(* CODESYS project BasePpt.library
   Company: Vistaprint
   Title: BasePpt
   Description: 0.0.0.10 - PCE: no EOFF State!! in EOFF go to OFF (in Always); Redo changes of 0.0.0.6; PTS.Always no EOFF; sta_OFFBusy in PTS reworked;
      0.0.0.9 - Merged the DeStacker MDC with the BasePpt MDC
      0.0.0.8 - Added newer Versions of libraries.
      0.0.0.7 - Added newer Versions of libraries.
      0.0.0.6 - Changes for Simualtion in MDC, sta_OFFBusy in PTB/MDC reworked; Always in PTB reworked;
      0.0.0.5 - Added new Base_PLC 0.3.4.1
      0.0.0.4 - Bug fixed in FB_PTB
      0.0.0.3 - Update to take the newest libraries 
      0.0.0.2 - Update to Base_PLC 0.3.3.2; Update to Base_Elements 0.0.0.9
   Author: pcipriano
   Version: 0.0.0.10

Project tree, tasks and I/O mapping:
  libraries: Base_Elements, 0.0.1.4 (Vistaprint); Base_PLC, 0.3.4.3 (Vistaprint); Tc2_Standard, 3.3.0.0 (Beckhoff Automation GmbH); Tc2_System, * (Beckhoff Automation GmbH); Tc2_Utilities, * (Beckhoff Automation GmbH); Tc3_Interfaces, 3.3.0.0 (Beckhoff Automation GmbH); Tc3_Module, * (Beckhoff Automation GmbH)
  POUs/
    Controller/
      Driver/
        PTR [Paper Tracker]/
          data type E_PTR_Status
          function block FB_PTR [ST]: BeltLength, EnterComplete, FB_init, Insert, PaperEntryOffset, PaperOnBelt, Pop, PositionList, Push, Reset, TimeBase
          data type T_PTR_STRUCT
      Lvl0/
      Lvl1/
        MDC [Malteser Drive Controller]/
          data type E_ALM_MDC
          function block FB_MDC [ST]: ActualPosition, Always, CtrlInit, CtrlSIf, Drive, FB_init, getCmdState, getCtrlSIf, GetTurningDirection, IncrementPosition, IoInBridge, IoOutBridge, SetPositionToGo, sta_ERROR, sta_ERRORQuit, sta_InitializeBusy, sta_InPosition, sta_InPositionBusy, sta_OFF, sta_OFFBusy, sta_PON, sta_PREPOSITION, sta_PREPOSITIONbusy, sta_StartTurnBusy, sta_TurnBusy, sta_TURNDONE, StateMachine
          global variables MDC_CmdState
          data type T_Ctrl_SIf_MDC
          data type T_Ctrl_SIf_MDC_Cfg
          data type T_Ctrl_SIf_MDC_Cur
          data type T_Ctrl_SIf_MDC_Ilk
          data type T_Ctrl_SIf_MDC_In
          data type T_Ctrl_SIf_MDC_Out
          data type T_Ctrl_SIf_MDC_Par
        PTB [Paper Transport Belt]/
          BeltParameterFunction/
            data type T_Belt_Cfg_Base
            data type T_Belt_Cur_Base
            data type T_Belt_Par_Base
          data type E_ALM_PTB
          data type E_BELT_DIRECTION
          data type E_PTB_MODE
          data type E_PTB_PaperDirection
          function block FB_PTB [ST]: Always, CalculateBeltParameter, CalculateModeParameter, CheckPumpState, cmd_OFF, cmd_RUN, cmd_STOP, CtrlInit, CtrlSIf, Drive, FB_init, getCmdState, getCtrlSIf, IoInBridge, IoOutBridge, PaperPositionHandling, PositionList, SetPumpComand, sta_EJECTPAPER, sta_EJECTPAPERbusy, sta_ERROR, sta_ERRORQuit, sta_OFF, sta_OFFBusy, sta_PON, sta_RUN, sta_RUNBusy, sta_STACKPAPER, sta_STACKPAPERbusy, sta_STOP, sta_STOPBusy, StateMachine, VacuumPump
          global variables PTB_CmdState
          data type T_Ctrl_SIf_PTB
          data type T_Ctrl_SIf_PTB_Cfg
          data type T_Ctrl_SIf_PTB_Cur
          data type T_Ctrl_SIf_PTB_Ilk
          data type T_Ctrl_SIf_PTB_In
          data type T_Ctrl_SIf_PTB_Out
          data type T_Ctrl_SIf_PTB_Par
      Lvl2/
        PBC [Paper Buffer Controller]/
          data type E_ALM_PBC
          function block FB_PBC [ST]: Always, Belt, CountPaper, CtrlInit, CtrlSIf, DeStacker, FB_init, getCmdState, getCtrlSIf, IoInBridge, IoOutBridge, PaperHight, PaperWidth, sta_EjectBusy, sta_EjectCheck, sta_ERROR, sta_ERRORQuit, sta_OFF, sta_OFFBusy, sta_PON, sta_PositionPaperBusy, sta_RUN, sta_RUNbusy, sta_STANDBY, sta_STANDBYBusy, StateMachine
          global variables PBC_CmdState
          data type T_Ctrl_SIf_PBC
          data type T_Ctrl_SIf_PBC_Cfg
          data type T_Ctrl_SIf_PBC_Cur
          data type T_Ctrl_SIf_PBC_Ilk
          data type T_Ctrl_SIf_PBC_In
          data type T_Ctrl_SIf_PBC_Out
          data type T_Ctrl_SIf_PBC_Par
        PCE [Paper Belt Corner Element]/
          data type E_ALM_PCE
          function block FB_PCE [ST]: Always, CtrlInit, CtrlSIf, DriveIn, DriveOut, FB_init, getCmdState, IoInBridge, IoOutBridge, PaperExitValveActive, PaperInputValveActive, sta_ERROR, sta_ERRORQuit, sta_OFF, sta_OFFBusy, sta_PON, sta_RUN, sta_RUNBusy, sta_STOP, sta_STOPBusy, StateMachine
          global variables PCE_CmdState
          data type T_Ctrl_SIf_PCE
          data type T_Ctrl_SIf_PCE_Cfg
          data type T_Ctrl_SIf_PCE_Cur
          data type T_Ctrl_SIf_PCE_Ilk
          data type T_Ctrl_SIf_PCE_In
          data type T_Ctrl_SIf_PCE_Out
          data type T_Ctrl_SIf_PCE_Par
      Lvl3/
        PTS [Paper Turning Station]/
          data type E_ALM_PTS
          data type E_PTS_MODE
          function block FB_PTS [ST]: Always, Belt, CalculateOutputDelay, CtrlInit, CtrlSIf, FB_init, getCmdState, getCtrlSIf, GetItemBusy, IoInBridge, IoOutBridge, Malteser, sta_EmptyDelayBusy, sta_ERROR, sta_ERRORQuit, sta_GetItemBusy, sta_InitializeBusy, sta_OFF, sta_OFFBusy, sta_PaperDelayBusy, sta_PON, sta_RUN, sta_RUNBusy, sta_STANDBY, sta_STANDBYBusy, sta_STOP, sta_STOPbusy, sta_TurnEmptyBusy, sta_TurnPaperBusy, sta_WaitPaper, sta_WaitPaperGone, StateMachine
          global variables PTS_CmdState
          data type T_Ctrl_SIf_PTS
          data type T_Ctrl_SIf_PTS_Cfg
          data type T_Ctrl_SIf_PTS_Cur
          data type T_Ctrl_SIf_PTS_Ilk
          data type T_Ctrl_SIf_PTS_In
          data type T_Ctrl_SIf_PTS_Out
          data type T_Ctrl_SIf_PTS_Par
          data type T_PTS_InOutPositions
      Lvl4/
      Top/
  Version/
    global variables Global_Version
*)

// POUs/Controller/Driver/PTR [Paper Tracker]/E_PTR_Status
TYPE E_PTR_Status :
(
	EnterBusy,
	OnBelt,
	ExitBusy,
	Gone,
	ERROR,
	MAX_E_PTR_Status
);
END_TYPE

// POUs/Controller/Driver/PTR [Paper Tracker]/T_PTR_STRUCT
TYPE T_PTR_STRUCT :
STRUCT
	// [us] Time of the paper on the belt
	udiTimeOnBelt_us				: UDINT;
	// [mm] Position of the paper on the belt
	lrePositionOnBelt_mm			: LREAL;
	// [mm] Position of the paper on the belt Adjusted to the possible maximum
	lrePositionOnBeltAdjusted_mm	: LREAL;
	// Paper Item Id
	udiItemId						: UDINT;
	// Error	
	eStatus							: E_PTR_Status;
END_STRUCT
END_TYPE

// POUs/Controller/Lvl1/MDC [Malteser Drive Controller]/E_ALM_MDC
TYPE E_ALM_MDC :
(
	TableSensorTimeout 		:= 1,
	CrossSensorTimeout		:= 2,
	PositionSame			:= 3,
	MAX_E_ALM_MDC
);
END_TYPE

// POUs/Controller/Lvl1/MDC [Malteser Drive Controller]/T_Ctrl_SIf_MDC
TYPE T_Ctrl_SIf_MDC :
STRUCT
	///configuration
	Cfg: T_Ctrl_SIf_MDC_Cfg;
	///parameter
	Par: T_Ctrl_SIf_MDC_Par;
	///current values
	Cur: T_Ctrl_SIf_MDC_Cur;
	///io input
	In: T_Ctrl_SIf_MDC_In;
	///io output
	Out: T_Ctrl_SIf_MDC_Out;
	///alarm number used in this controller
	Alm: ARRAY[1..MAX_E_ALM_MDC] OF T_Ctrl_Alm;
	///interlock of output/movements
	Ilk: T_Ctrl_SIf_MDC_Ilk;
END_STRUCT
END_TYPE

// POUs/Controller/Lvl1/MDC [Malteser Drive Controller]/T_Ctrl_SIf_MDC_Cfg
TYPE T_Ctrl_SIf_MDC_Cfg :
STRUCT
	/// Number of positions in 360° of the Malteser drive
	uintPositionPerTurn		: UINT;
END_STRUCT
END_TYPE

// POUs/Controller/Lvl1/MDC [Malteser Drive Controller]/T_Ctrl_SIf_MDC_Cur
TYPE T_Ctrl_SIf_MDC_Cur :
STRUCT	
	/// Actual Position as position 
	uintActualPosition			: UINT;
	/// actual turning direction
	eActualTurningDirection		: E_TURN_DIRECTION;
	/// Reference still ok
	bolReferenceOk				: BOOL;		
END_STRUCT
END_TYPE

// POUs/Controller/Lvl1/MDC [Malteser Drive Controller]/T_Ctrl_SIf_MDC_Ilk
TYPE T_Ctrl_SIf_MDC_Ilk :
STRUCT
END_STRUCT
END_TYPE

// POUs/Controller/Lvl1/MDC [Malteser Drive Controller]/T_Ctrl_SIf_MDC_In
TYPE T_Ctrl_SIf_MDC_In :
STRUCT
	/// Is the cross in sensor positinon. One rotation step done.
	bolCrossPositionSensor				: BASE_PLC.T_Ctrl_IoBool;
	/// Is the table at 0° degrees
	bolTablePositionSensor				: BASE_PLC.T_Ctrl_IoBool;
END_STRUCT
END_TYPE

// POUs/Controller/Lvl1/MDC [Malteser Drive Controller]/T_Ctrl_SIf_MDC_Out
TYPE T_Ctrl_SIf_MDC_Out :
STRUCT
	intActualPosition		: BASE_PLC.T_Ctrl_IoInt;
END_STRUCT
END_TYPE

// POUs/Controller/Lvl1/MDC [Malteser Drive Controller]/T_Ctrl_SIf_MDC_Par
TYPE T_Ctrl_SIf_MDC_Par :
STRUCT
	/// <0 = Turn left; =0 automatic; >0 turn right
	intTurnDirection					: INT;
	/// Position to go to if comand turn is given. 0 = initialization position
	uinPositionToGo						: UINT;
	/// [ms] time to rotate one step 
	udiStepRotationTime_ms				: UDINT;
	/// [ms] initialization timeout time
	udiInitializationTime_ms			: UDINT;
	/// [ms] simulation time to rotate one step
	udiSimStepRotationTime_ms			: UDINT;
	/// [ms] simulation initialization timeout time
	udiSimInitializationTime_ms			: UDINT;
	/// [ms] simulation time to start rotate and Cross sensor needs to go away
	udiSimStartRotationTime_ms			: UDINT;
	/// [rpm] PrePosition Speed
	uinPrePositionSpeed_rpm				: UINT;
	/// [rpm] Position Speed
	uinPositionSpeed_rpm				: UINT;
END_STRUCT
END_TYPE

// POUs/Controller/Lvl1/PTB [Paper Transport Belt]/BeltParameterFunction/T_Belt_Cfg_Base
TYPE T_Belt_Cfg_Base :
STRUCT
	/// Assign the motor rotation to a belt direction.
	intForwardDirection				: INT;
	/// Assign the motor rotation to a belt direction.
	intBackwardDirection			: INT;
	/// [mm] the belt travels per motor rotation
	reaRpmDistance_mm					: REAL;
END_STRUCT
END_TYPE

// POUs/Controller/Lvl1/PTB [Paper Transport Belt]/BeltParameterFunction/T_Belt_Cur_Base
TYPE T_Belt_Cur_Base :
STRUCT
	/// [mm/s] Belt speed
	uinBeltSpeed_mms						: UINT;
	/// [rpm] Belt speed
	uinBeltSpeed_rpm						: UINT;
END_STRUCT
END_TYPE

// POUs/Controller/Lvl1/PTB [Paper Transport Belt]/BeltParameterFunction/T_Belt_Par_Base
TYPE T_Belt_Par_Base :
STRUCT
	/// eSpeedControlSelection.EFFECTIVE_SPEED : [mm/sec] Target speed. Uses reaRpmDistance_mm and uinLC11 to calculate the rpm
	uinBeltSpeed						: UINT;
	/// eSpeedControlSelection.EFFECTIVE_SPEED : [mm/sec] Target speed. Uses reaRpmDistance_mm and uinLC11 to calculate the rpm
	uinStackSpeed						: UINT;
END_STRUCT
END_TYPE

// POUs/Controller/Lvl1/PTB [Paper Transport Belt]/E_ALM_PTB
TYPE E_ALM_PTB :
(
	TestAlarm := 1,
	MAX_E_ALM_PTB 
);
END_TYPE

// POUs/Controller/Lvl1/PTB [Paper Transport Belt]/E_BELT_DIRECTION
TYPE E_BELT_DIRECTION :
(
	FORWARD			:= 0,
	BACKWARD		:= 1,
	MAX_E_BELT_DIRECTION
);
END_TYPE

// POUs/Controller/Lvl1/PTB [Paper Transport Belt]/E_PTB_MODE
TYPE E_PTB_MODE :
(
	Endless	,		// 0
	ToSensor,		// 1
	ToDistance,		// 2
	ToTime,			// 3
	Stack,			// 4
	MAX_E_PTB_MODE
);
END_TYPE

// POUs/Controller/Lvl1/PTB [Paper Transport Belt]/E_PTB_PaperDirection
TYPE E_PTB_PaperDirection :
(
	Portrait,
	Landscape,
	MAX_E_PTB_PaperDirection
);
END_TYPE

// POUs/Controller/Lvl1/PTB [Paper Transport Belt]/T_Ctrl_SIf_PTB
TYPE T_Ctrl_SIf_PTB :
STRUCT
	///configuration
	Cfg: T_Ctrl_SIf_PTB_Cfg;
	///parameter
	Par: T_Ctrl_SIf_PTB_Par;
	///current values
	Cur: T_Ctrl_SIf_PTB_Cur;
	///io input
	In: T_Ctrl_SIf_PTB_In;
	///io output
	Out: T_Ctrl_SIf_PTB_Out;
	///alarm number used in this controller
	Alm: ARRAY[1..E_ALM_PTB.MAX_E_ALM_PTB] OF T_Ctrl_Alm;
	///interlock of output/movements
	Ilk: T_Ctrl_SIf_PTB_Ilk;
END_STRUCT
END_TYPE

// POUs/Controller/Lvl1/PTB [Paper Transport Belt]/T_Ctrl_SIf_PTB_Cfg
TYPE T_Ctrl_SIf_PTB_Cfg :
STRUCT
	// Function Mode
	eMode							: E_PTB_MODE;
	// Vacuum pump present
	bolVacuumPresent				: BOOL;
	// [mm] Length of the belt
	udiBeltLength_mm				: UDINT;
	// Belt Parameter	
	rBeltParam						: T_Belt_Cfg_Base;
	// Enable Entry Belt Sensor Debounce
	bolEntrySensorDebounceEnable	: BOOL;
	// Enable Exit Belt Sensor Debounce
	bolExitSensorDebounceEnable		: BOOL;
END_STRUCT
END_TYPE

// POUs/Controller/Lvl1/PTB [Paper Transport Belt]/T_Ctrl_SIf_PTB_Cur
	TYPE T_Ctrl_SIf_PTB_Cur :
STRUCT	
	/// actual belt direction
	eActualDirection						: E_BELT_DIRECTION;
	/// [mm] Distance to move if Move Mode is distance
	udiDistanceToMove_mm					: UDINT;
	/// [ms] Time to move
	udiTimeToMove_ms						: UDINT;
	// Belt parameter
	rBeltParam								: T_Belt_Cur_Base;
	// Belt Run Time
	udiBeltTimeBase_mm						: UDINT;
	// Paper on the belt
	uinPaperOnBelt							: UINT;
	// Pointer to the Position list of the paper on the belt
	pPositionList							: POINTER TO T_PTR_STRUCT;
END_STRUCT
END_TYPE

// POUs/Controller/Lvl1/PTB [Paper Transport Belt]/T_Ctrl_SIf_PTB_Ilk
TYPE T_Ctrl_SIf_PTB_Ilk :
STRUCT
END_STRUCT
END_TYPE

// POUs/Controller/Lvl1/PTB [Paper Transport Belt]/T_Ctrl_SIf_PTB_In
TYPE T_Ctrl_SIf_PTB_In :
STRUCT
	bolBeltEntrySensor			: BASE_PLC.T_Ctrl_IoBool;
	bolBeltExitSensor			: BASE_PLC.T_Ctrl_IoBool;
	bolBeltEntrySensorPEdge		: BASE_PLC.T_Ctrl_IoBool;
	bolBeltEntrySensorNEdge		: BASE_PLC.T_Ctrl_IoBool;
	bolBeltExitSensorPEdge		: BASE_PLC.T_Ctrl_IoBool;
	bolBeltExitSensorNEdge		: BASE_PLC.T_Ctrl_IoBool;
END_STRUCT
END_TYPE

// POUs/Controller/Lvl1/PTB [Paper Transport Belt]/T_Ctrl_SIf_PTB_Out
TYPE T_Ctrl_SIf_PTB_Out :
STRUCT

END_STRUCT
END_TYPE

// POUs/Controller/Lvl1/PTB [Paper Transport Belt]/T_Ctrl_SIf_PTB_Par
TYPE T_Ctrl_SIf_PTB_Par :
STRUCT
	/// <0 = Backward; =0 None; >0 forward
	intDirection						: INT;
	/// [mm] Distance to move if Move Mode is distance
	udiDistanceToMove_mm				: UDINT;
	/// [ms] Time to move
	udiTimeToMove_ms					: UDINT;
	/// Stack hight in # of sheets
	uinPaperStackHight					: UINT;
	/// Automatic ejecting the paper if stackhight is reached
	bolAutoEjectAfterStack				: BOOL;
	/// Automatic stacking the paper after ejecting all paper
	bolAutoStackAfterEject				: BOOL;
	/// Belt Parameter
	rBeltParam							: T_Belt_Par_Base;
	// [ms] Stack delay time - Delay before out motor can move after paper entered system
	udiStackDelayTime_ms				: UDINT;
	// [mm] Belt Length
	udiBeltLength_mm					: UDINT;
	// Page running format
	ePaperOrientation					: E_PTB_PaperDirection;
	/// [mm] Paper Hight
	uinPaperHight_mm					: UINT;
	/// [mm] Paper Width
	uinPaperWidth_mm					: UINT;
	// [ms] Input Parameter Debounce time
	uinInputSignalDebounceTime_ms		: UINT;
END_STRUCT
END_TYPE

// POUs/Controller/Lvl2/PBC [Paper Buffer Controller]/E_ALM_PBC
TYPE E_ALM_PBC :
(
	PaperTransport			:= 1,
	BufferFull				:= 2,
	BufferEmpty				:= 3,
	MAX_E_ALM_PBC
);
END_TYPE

// POUs/Controller/Lvl2/PBC [Paper Buffer Controller]/T_Ctrl_SIf_PBC
TYPE T_Ctrl_SIf_PBC :
STRUCT
	///configuration
	Cfg: T_Ctrl_SIf_PBC_Cfg;
	///parameter
	Par: T_Ctrl_SIf_PBC_Par;
	///current values
	Cur: T_Ctrl_SIf_PBC_Cur;
	///io input
	In: T_Ctrl_SIf_PBC_In;
	///io output
	Out: T_Ctrl_SIf_PBC_Out;
	///alarm number used in this controller
	Alm: ARRAY[1..E_ALM_PBC.MAX_E_ALM_PBC] OF T_Ctrl_Alm;
	///interlock of output/movements
	Ilk: T_Ctrl_SIf_PBC_Ilk;
END_STRUCT
END_TYPE

// POUs/Controller/Lvl2/PBC [Paper Buffer Controller]/T_Ctrl_SIf_PBC_Cfg
TYPE T_Ctrl_SIf_PBC_Cfg :
STRUCT
END_STRUCT
END_TYPE

// POUs/Controller/Lvl2/PBC [Paper Buffer Controller]/T_Ctrl_SIf_PBC_Cur
TYPE T_Ctrl_SIf_PBC_Cur :
STRUCT	
	/// How many papers are in the buffer. -1 = Paper count unknown
	uinPaperInBufferCount			: UINT;
	/// Last Paper to eject count parameter
	uinPaperToEjectParameter		: UINT;
	/// Actual count of the paper ejected 
	uinPaperToEjectCount			: UINT;
	/// [ms] Time from sheet to sheet ejection in multi eject mode.
	uinSheetToSheetTime				: UINT;
	// Was paper before Eject available
	bolPaperBeforeEjectAvailable	: BOOL;
	// Paper to paper Timeout
	uinPaperToPaperTime_ms			: UINT;
END_STRUCT
END_TYPE

// POUs/Controller/Lvl2/PBC [Paper Buffer Controller]/T_Ctrl_SIf_PBC_Ilk
TYPE T_Ctrl_SIf_PBC_Ilk :
STRUCT
END_STRUCT
END_TYPE

// POUs/Controller/Lvl2/PBC [Paper Buffer Controller]/T_Ctrl_SIf_PBC_In
TYPE T_Ctrl_SIf_PBC_In :
STRUCT
	/// This sensor shows if the buffer reaches his capacity limits
	bolPaperAvailableExit					: BASE_PLC.T_Ctrl_IoBool;
	/// Shows if there is paper available in the buffer
	bolPaperAvailableEntry					: BASE_PLC.T_Ctrl_IoBool;
	/// Shows if there is a paper on the output of the buffer
	bolCapacityReached						: BASE_PLC.T_Ctrl_IoBool;
END_STRUCT
END_TYPE

// POUs/Controller/Lvl2/PBC [Paper Buffer Controller]/T_Ctrl_SIf_PBC_Out
TYPE T_Ctrl_SIf_PBC_Out :
STRUCT
END_STRUCT
END_TYPE

// POUs/Controller/Lvl2/PBC [Paper Buffer Controller]/T_Ctrl_SIf_PBC_Par
TYPE T_Ctrl_SIf_PBC_Par :
STRUCT
	/// [ms] Paper transport timeout - Time that paper is allowed to have for the transport to the front.
	udiPaperTransportTime				: UDINT;
	/// Sheet to output with one run command.  0 = endless until stop
	udiSheetToEject						: UDINT;
	/// [ms] Time from sheet to sheet ejection in multi eject mode.
	udiSheetToSheetTime					: UDINT;
	/// [ms] Paper transport time simulation
	udiSimPaperTransportTime			: UDINT;
	/// [ms] Paper to paper transport time simulation
	udiSimPaperToPaperTransportTime		: UDINT;
END_STRUCT
END_TYPE

// POUs/Controller/Lvl2/PCE [Paper Belt Corner Element]/E_ALM_PCE
TYPE E_ALM_PCE :
(
	PaperSensorError := 1,
	MAX_E_ALM_PCE 
);
END_TYPE

// POUs/Controller/Lvl2/PCE [Paper Belt Corner Element]/T_Ctrl_SIf_PCE
TYPE T_Ctrl_SIf_PCE :
STRUCT
	///configuration
	Cfg: T_Ctrl_SIf_PCE_Cfg;
	///parameter
	Par: T_Ctrl_SIf_PCE_Par;
	///current values
	Cur: T_Ctrl_SIf_PCE_Cur;
	///io input
	In: T_Ctrl_SIf_PCE_In;
	///io output
	Out: T_Ctrl_SIf_PCE_Out;
	///alarm number used in this controller
	Alm: ARRAY[1..MAX_E_ALM_PCE] OF T_Ctrl_Alm;
	///interlock of output/movements
	Ilk: T_Ctrl_SIf_PCE_Ilk;
END_STRUCT
END_TYPE

// POUs/Controller/Lvl2/PCE [Paper Belt Corner Element]/T_Ctrl_SIf_PCE_Cfg
TYPE T_Ctrl_SIf_PCE_Cfg :
STRUCT
END_STRUCT
END_TYPE

// POUs/Controller/Lvl2/PCE [Paper Belt Corner Element]/T_Ctrl_SIf_PCE_Cur
TYPE T_Ctrl_SIf_PCE_Cur :
STRUCT	
	/// [mm/s] Belt speed
	uinBeltSpeed					: UINT;
END_STRUCT
END_TYPE

// POUs/Controller/Lvl2/PCE [Paper Belt Corner Element]/T_Ctrl_SIf_PCE_Ilk
TYPE T_Ctrl_SIf_PCE_Ilk :
STRUCT
END_STRUCT
END_TYPE

// POUs/Controller/Lvl2/PCE [Paper Belt Corner Element]/T_Ctrl_SIf_PCE_In
TYPE T_Ctrl_SIf_PCE_In :
STRUCT
	/// 0 = Paper not here; 1 = Paper detected
	bolPaperAvailable				: BASE_PLC.T_Ctrl_IoBool;
END_STRUCT
END_TYPE

// POUs/Controller/Lvl2/PCE [Paper Belt Corner Element]/T_Ctrl_SIf_PCE_Out
TYPE T_Ctrl_SIf_PCE_Out :
STRUCT
	/// Paper Incoming Belt - 0 = Vacuum Valve Closed;  1 = Vacuum valve open
	bolVacuumValveIn 			: BASE_PLC.T_Ctrl_IoBool;
	/// Paper Outgoing Belt - 0 = Vacuum Valve Closed;  1 = Vacuum valve open
	bolVacuumValveOut 			: BASE_PLC.T_Ctrl_IoBool;
END_STRUCT
END_TYPE

// POUs/Controller/Lvl2/PCE [Paper Belt Corner Element]/T_Ctrl_SIf_PCE_Par
TYPE T_Ctrl_SIf_PCE_Par :
STRUCT
	/// [ms] Paper entry delay time. Time delay between detection and switching the vacuum
	uinPaperEntryDelayTime_ms		:UDINT;
	/// [ms] Paper exit time
	uinPaperExitTime_ms				:UDINT;
	/// [ms] Simulation Paper exit time
	uinSimPaperExitTime_ms			:UDINT;
END_STRUCT
END_TYPE

// POUs/Controller/Lvl3/PTS [Paper Turning Station]/E_ALM_PTS
TYPE E_ALM_PTS :
(
	PaperTransport			:= 1,
	ModeParameter			:= 2,
	MAX_E_ALM_PTS
);
END_TYPE

// POUs/Controller/Lvl3/PTS [Paper Turning Station]/E_PTS_MODE
TYPE E_PTS_MODE :
(
	Automatic 	:= -2,
	Distribute	:= -1,
	FixA		:= 0,
	FixB		:= 1,
	FixC		:= 2,
	MAX_E_PTS_MODE
);
END_TYPE

// POUs/Controller/Lvl3/PTS [Paper Turning Station]/T_Ctrl_SIf_PTS
TYPE T_Ctrl_SIf_PTS :
STRUCT
	///configuration
	Cfg: T_Ctrl_SIf_PTS_Cfg;
	///parameter
	Par: T_Ctrl_SIf_PTS_Par;
	///current values
	Cur: T_Ctrl_SIf_PTS_Cur;
	///io input
	In: T_Ctrl_SIf_PTS_In;
	///io output
	Out: T_Ctrl_SIf_PTS_Out;
	///alarm number used in this controller
	Alm: ARRAY[1..MAX_E_ALM_PTS] OF T_Ctrl_Alm;
	///interlock of output/movements
	Ilk: T_Ctrl_SIf_PTS_Ilk;
END_STRUCT
END_TYPE

// POUs/Controller/Lvl3/PTS [Paper Turning Station]/T_Ctrl_SIf_PTS_Cfg
TYPE T_Ctrl_SIf_PTS_Cfg :
STRUCT
	// Turns the barcode reader intelligence on. This makes the PTS nearly self sustained. 
	bolBarcodeReaderAvailable			: BOOL;
	// If there is no barcode but a sensor at the end of the entry belt 
	bolEntrySensorAvailable				: BOOL;
	// Paper Input and Ouput Positions for the fixed modes
	aFixPosDef							: ARRAY[0..E_PTS_MODE.MAX_E_PTS_MODE-1] OF T_PTS_InOutPositions;
	// Automatic Mode Input and Output Positions
	aAutoPosDef							: ARRAY[0..cPTS_MAX_AUTOPOS-1] OF T_PTS_InOutPositions;
	// Automatic Mode Default Input Positions
	aDefaultAutoPos						: UINT;
	// Paper Input and Ouput Positions for the fixed modes
	aDistributionPositionDefinition		: ARRAY[0..PTS_CmdState.cPTS_MAX_DISTRIBUTION-1] OF E_PTS_MODE;
	// Start positioning the malteser wheel before turning
	bolPositionMalteserEnable			: BOOL;
END_STRUCT
END_TYPE

// POUs/Controller/Lvl3/PTS [Paper Turning Station]/T_Ctrl_SIf_PTS_Cur
TYPE T_Ctrl_SIf_PTS_Cur :
STRUCT	
	/// Actual Sheet In- Out- Positions
	rInOutPosition					: T_PTS_InOutPositions;
	/// Saves the last executed distribution index
	iActualDistributionIndex		: INT;
	/// [ms] Time to wait after paper was detected before to turn.
	udiPaperInTurnDelayTime				: UDINT;
	/// [ms] Time to wait after paper is not detected anymore before to turn back.
	udiPaperOutTurnDelayTime			: UDINT;
END_STRUCT
END_TYPE

// POUs/Controller/Lvl3/PTS [Paper Turning Station]/T_Ctrl_SIf_PTS_Ilk
TYPE T_Ctrl_SIf_PTS_Ilk :
STRUCT
END_STRUCT
END_TYPE

// POUs/Controller/Lvl3/PTS [Paper Turning Station]/T_Ctrl_SIf_PTS_In
TYPE T_Ctrl_SIf_PTS_In :
STRUCT
	/// This sensor shows if the paper is at the middle table possition
	bolPaperAvailable   					: BASE_PLC.T_Ctrl_IoBool;
	/// This sensor shows if the paper is available at the exit of the input belt
	bolPaperAtBeltExit						: BASE_PLC.T_Ctrl_IoBool;
END_STRUCT
END_TYPE

// POUs/Controller/Lvl3/PTS [Paper Turning Station]/T_Ctrl_SIf_PTS_Out
TYPE T_Ctrl_SIf_PTS_Out :
STRUCT
END_STRUCT
END_TYPE

// POUs/Controller/Lvl3/PTS [Paper Turning Station]/T_Ctrl_SIf_PTS_Par
TYPE T_Ctrl_SIf_PTS_Par :
STRUCT
	/// [ms] Time to wait after paper was detected before to turn.
	udiPaperInTurnDelayTime				: UDINT;
	/// [ms] Time to wait after paper is not detected anymore before to turn back.
	udiPaperOutTurnDelayTime			: UDINT;
	/// [ms] Timeout for the time the Paper can have between Barcode reader and Paper on table sensor.
	udiPaperBarcodeToInputSensorTime	: UDINT;
	/// Mode for turning
	eMode								: E_PTS_MODE;
	/// [ms] Simulation Timeout for the time the Paper can have between Barcode reader and Paper on table sensor.
	udiSimPaperBarcodeToInputSensorTime	: UDINT;
END_STRUCT
END_TYPE

// POUs/Controller/Lvl3/PTS [Paper Turning Station]/T_PTS_InOutPositions
TYPE T_PTS_InOutPositions :
STRUCT
	uinInput			: UINT;
	uinOutput			: UINT;
	eDirection			: E_TURN_DIRECTION;
END_STRUCT
END_TYPE

// POUs/Controller/Lvl1/MDC [Malteser Drive Controller]/MDC_CmdState
VAR_GLOBAL CONSTANT
	///ctrl commands definitions
	///specific commands >200 - every command has to be a even number
	cCMD_INITIALIZE			: INT := 202;
	cCMD_TURN    			: INT := 204;
	cCMD_PREPOSITION		: INT := 210;
	
	///ctrl specific states definitions
	cSTA_InitializeBusy		: INT := 201;
	cSTA_InPositionBusy		: INT := 203;
	cSTA_InPosition			: INT := 205;
	cSTA_StartTurnBusy		: INT := 207;
	cSTA_TurnBusy			: INT := 209;
	cSTA_PREPOSITIONbusy	: INT := 220;
	cSTA_PREPOSITION		: INT := 221;
	cSTA_TURNDONE			: INT := 222;
	
	cSUB_TURNbusy			: INT := 300;
	cSUB_STOPbusy			: INT := 301;
	cSUB_FINDHOLEbusy		: INT := 302;
END_VAR

// POUs/Controller/Lvl1/PTB [Paper Transport Belt]/PTB_CmdState
VAR_GLOBAL CONSTANT
	///ctrl commands definitions
	cCMD_EJECTPAPER			: INT := 202;
	cCMD_STACKPAPER			: INT := 204;
	///specific commands >200 - every command has to be a even number
	///ctrl specific states definitions
	cSTA_EJECTPAPERbusy		: INT := 201;
	cSTA_EJECTPAPER			: INT := 202;
	cSTA_STACKPAPERbusy		: INT := 203;
	cSTA_STACKPAPER			: INT := 204;

	///ctrl specific sub states definitions
	cSUB_EMPTYstart					: INT := 300;
	cSUB_EMPTYWAITPAPERbusy			: INT := 301;
	cSUB_EMPTYWAITPAPERdebounce		: INT := 302;
	cSUB_EMPTYWAITPAPERGONEbusy		: INT := 303;
	cSUB_EMPTYWAITPAPERGONEdebounce	: INT := 304;
	cSUB_EMPTYWAITDRIVESTOPED		: INT := 305;
	cSUB_WAITPAPER  				: INT := 306;
	cSUB_WAITPAPERGONE  			: INT := 307;
	cSUB_STARTSTACKDELAY			: INT := 308;
	cSUB_PAPERDISTANCEstart			: INT := 309;
	cSUB_PAPERDISTANCEbusy			: INT := 310;
	cSUB_PAPERDISTANCESTOPbusy		: INT := 311;
	cSUB_STARTENTRYDRIVEbusy		: INT := 312;
	cSUB_STARTENTRYDRIVE			: INT := 313;
END_VAR

// POUs/Controller/Lvl2/PBC [Paper Buffer Controller]/PBC_CmdState
VAR_GLOBAL CONSTANT
	///ctrl specific command definitions
	cCMD_SINGLE				: INT := 202;
	cCMD_STANDBY			: INT := 204;
	
	///ctrl specific states definitions
	cSTA_STANDBYBusy		: INT := 203;
	cSTA_STANDBY			: INT := 204;
	cSTA_PositionPaperBusy	: INT := 205;
	cSTA_RUNEmpty			: INT := 207;
	cSTA_EjectBusy			: INT := 209;
	cSTA_EjectCheck			: INT := 211;
	
	cSUB_WAITPAPER			: INT := 300;
	cSUB_POSITIONbusy		: INT := 301;
	cSUB_POSITIONSTOPbusy	: INT := 302;
	cSUB_EVALUATEEJECT		: INT := 303;
	cSUB_EJECTbusy			: INT := 304;
	cSUB_EJECTSTOPbusy		: INT := 305;
	cSUB_POSITIONSTARTbusy	: INT := 306;
	cSUB_EJECTSTARTbusy		: INT := 307;
	cSUB_READYEJECT			: INT := 308;
	
//	cSUB_WAITPAPER
END_VAR

// POUs/Controller/Lvl2/PCE [Paper Belt Corner Element]/PCE_CmdState
VAR_GLOBAL CONSTANT
	///ctrl commands definitions
	///specific commands >200 - every command has to be a even number
	///ctrl specific states definitions
	cSUB_PAPERENTRY				: INT := 300;
	cSUB_PAPERENTRYDelay		: INT := 301;
	cSUB_PAPEREXIT				: INT := 302;
END_VAR

// POUs/Controller/Lvl3/PTS [Paper Turning Station]/PTS_CmdState
VAR_GLOBAL CONSTANT
	///ctrl specific command definitions
	cCMD_TURN				: INT := 202;
	cCMD_STANDBY			: INT := 204;
	
	///ctrl specific states definitions
	cSTA_STANDBYBusy		: INT := 203;
	cSTA_STANDBY			: INT := 204;
	cSTA_PaperDelayBusy  	: INT := 205;
	cSTA_TurnPaperBusy		: INT := 207;
	cSTA_WaitPaperGone		: INT := 209;
	cSTA_EmptyDelayBusy		: INT := 211;
	cSTA_TurnEmptyBusy		: INT := 213;
	cSTA_InitializeBusy		: INT := 215;
	cSTA_WaitPaper			: INT := 217;
	cSTA_GetItemBusy		: INT := 219;
	
	// ctrl specific substates definitions
	cSUB_WAIT_START			: INT := 300;
	cSUB_WAIT_DONE 			: INT := 301;
	cSUB_TURNbusy			: INT := 302;
	cSUB_TURNDONE			: INT := 303;
	cSUB_PREPOSITIONbusy	: INT := 304;
	
	// Other Constants
	cPTS_MAX_AUTOPOS		: UINT	:= 5;
	cPTS_MAX_DISTRIBUTION	: INT	:= 2;
END_VAR

// Version/Global_Version
// This function has been automatically generated from the project information.
VAR_GLOBAL CONSTANT
	{attribute 'const_non_replaced'}
	stLibVersion_BasePpt : ST_LibVersion := (iMajor := 0, iMinor := 0, iBuild := 0, iRevision := 10, sVersion := '0.0.0.10');
END_VAR

// POUs/Controller/Driver/PTR [Paper Tracker]/FB_PTR
FUNCTION_BLOCK PUBLIC FB_PTR
VAR_INPUT
	In_uinBeltSpeed		: UINT;
END_VAR
VAR_OUTPUT
END_VAR
VAR
	m_udiTimeBase_us			: UDINT;		// Time base in [usec]
	m_intPaperOnBelt			: INT;			// # of Paper on the belt 
	m_intFirstPaperIdx			: INT;			// Index of the leading paper on the belt
	m_intLastPaperIdx			: INT;			// Index of the last paper on the belt
	m_arBuffer					: ARRAY[0..THIS^.cMAXBUFFERSIZE-1] OF T_PTR_STRUCT;
	m_arPositionList			: ARRAY[0..THIS^.cMAXBUFFERSIZE-1] OF T_PTR_STRUCT;
	m_intPaperEntryOffset_mm	: INT;
	m_dinBeltLength				: DINT;
	
	iIdx					: INT;
	iNdx					: INT;
	iDifference				: DINT;
END_VAR
VAR CONSTANT
	cMAXBUFFERSIZE					: INT  := 20;
	cPAPERPOSITION_TOLERANCE_mm		: UINT := 200;
END_VAR

IF m_intPaperOnBelt > 0 THEN
	iNdx := m_intFirstPaperIdx;
	
	FOR iIdx := 0 TO m_intPaperOnBelt-1 DO
		m_arBuffer[iNdx].udiTimeOnBelt_us := m_arBuffer[iNdx].udiTimeOnBelt_us + THIS^.m_udiTimeBase_us;
		m_arBuffer[iNdx].lrePositionOnBelt_mm := m_arBuffer[iNdx].lrePositionOnBelt_mm + UDINT_TO_LREAL(THIS^.m_udiTimeBase_us) * UDINT_TO_LREAL(THIS^.In_uinBeltSpeed) / 1000000.0;
				
		CASE m_arBuffer[iNdx].eStatus OF
			E_PTR_Status.EnterBusy:
				m_arBuffer[iNdx].lrePositionOnBeltAdjusted_mm := MIN(m_intPaperEntryOffset_mm, LREAL_TO_INT(m_arBuffer[iNdx].lrePositionOnBelt_mm));
				iDifference := m_intPaperEntryOffset_mm - LREAL_TO_DINT(m_arBuffer[iNdx].lrePositionOnBelt_mm);
					
				IF 	(iDifference < 0) AND (ABS(iDifference) > cPAPERPOSITION_TOLERANCE_mm) THEN
					m_arBuffer[iNdx].eStatus := E_PTR_Status.ERROR;
				END_IF
			E_PTR_Status.OnBelt:
				m_arBuffer[iNdx].lrePositionOnBeltAdjusted_mm := MIN(m_dinBeltLength, LREAL_TO_DINT(m_arBuffer[iNdx].lrePositionOnBelt_mm));
				iDifference := m_dinBeltLength - LREAL_TO_DINT(m_arBuffer[iNdx].lrePositionOnBelt_mm);

				IF 	(iDifference < 0) AND (ABS(iDifference) > cPAPERPOSITION_TOLERANCE_mm) THEN
					m_arBuffer[iNdx].eStatus :=  E_PTR_Status.ERROR;
				END_IF
			E_PTR_Status.ExitBusy:
		END_CASE
		
		m_arPositionList[iIdx] :=  m_arBuffer[iNdx];	
		iNdx := (iNdx + 1) MOD THIS^.cMAXBUFFERSIZE;
	END_FOR
ELSE
	m_arPositionList[0].eStatus := E_PTR_Status.Gone;
END_IF

PROPERTY PUBLIC BeltLength : DINT
GET
BeltLength := m_dinBeltLength;
END_GET
SET
m_dinBeltLength := BeltLength;
END_SET
END_PROPERTY

METHOD PUBLIC EnterComplete : BOOL
VAR_INPUT
END_VAR
m_arBuffer[m_intLastPaperIdx].eStatus := E_PTR_Status.OnBelt;
m_arBuffer[m_intLastPaperIdx].lrePositionOnBelt_mm := INT_TO_LREAL(m_intPaperEntryOffset_mm);
m_arBuffer[m_intLastPaperIdx].lrePositionOnBeltAdjusted_mm := INT_TO_LREAL(m_intPaperEntryOffset_mm);
END_METHOD

METHOD FB_init : BOOL
VAR_INPUT
	bInitRetains : BOOL; // if TRUE, the retain variables are initialized (warm start / cold start)
	bInCopyCode : BOOL;  // if TRUE, the instance afterwards gets moved into the copy code (online change)
END_VAR
m_udiTimeBase_us := 2000;
m_intPaperEntryOffset_mm := 0;
Reset();
END_METHOD

METHOD PUBLIC Insert : BOOL
VAR_INPUT
	uinPosition_mm			: UINT;
	udiItemId				: UDINT;
END_VAR
VAR
	iIdx					: INT;
	iNdx					: INT;
	iInsertIdx				: INT;
END_VAR
iInsertIdx := m_intFirstPaperIdx;
iNdx := m_intFirstPaperIdx;
iIdx := 0;
	
WHILE (iIdx < m_intPaperOnBelt) AND (uinPosition_mm < m_arBuffer[iNdx].lrePositionOnBelt_mm) DO
	iIdx := iIdx + 1;
	iNdx := (iNdx + 1) MOD THIS^.cMAXBUFFERSIZE;
END_WHILE
END_METHOD

PROPERTY PUBLIC PaperEntryOffset : INT
GET
PaperEntryOffset := m_intPaperEntryOffset_mm;
END_GET
SET
m_intPaperEntryOffset_mm := PaperEntryOffset;
END_SET
END_PROPERTY

PROPERTY PUBLIC PaperOnBelt : UINT
GET
PaperOnBelt := INT_TO_UINT(m_intPaperOnBelt);
END_GET
SET
END_SET
END_PROPERTY

METHOD PUBLIC Pop : T_PTR_STRUCT
// Remove a paper from the buffer
VAR_INPUT
END_VAR
Pop.eStatus := E_PTR_Status.Gone;
Pop.lrePositionOnBelt_mm := 0.0;
Pop.lrePositionOnBeltAdjusted_mm := 0.0;
Pop.udiItemId := 0;
Pop.udiTimeOnBelt_us := 0;


IF m_intPaperOnBelt > 0 THEN
	Pop := m_arBuffer[m_intFirstPaperIdx];
	m_arBuffer[m_intFirstPaperIdx].udiItemId := 0;
	m_arBuffer[m_intFirstPaperIdx].lrePositionOnBelt_mm := 0.0;
	m_arBuffer[m_intFirstPaperIdx].lrePositionOnBeltAdjusted_mm := 0.0;
	m_arBuffer[m_intFirstPaperIdx].udiTimeOnBelt_us := 0;
	m_arBuffer[m_intFirstPaperIdx].eStatus := E_PTR_Status.Gone;
	m_intPaperOnBelt := m_intPaperOnBelt - 1;

	IF m_intPaperOnBelt = 0 THEN
		m_arPositionList[0] := m_arBuffer[m_intFirstPaperIdx];
	END_IF

	m_intFirstPaperIdx := (m_intFirstPaperIdx + 1) MOD THIS^.cMAXBUFFERSIZE;
END_IF
END_METHOD

PROPERTY PUBLIC PositionList : POINTER TO T_PTR_STRUCT
GET
VAR
	iIdx			: INT;
	iNdx			: INT;
END_VAR
PositionList := ADR(m_arPositionList);
END_GET
SET
END_SET
END_PROPERTY

METHOD PUBLIC Push : BOOL
// Add (Push) a paper into the buffer
// Return an ID for the paper
VAR_INPUT
	In_udiItemId			: UDINT;
END_VAR
Push := FALSE;

IF m_intPaperOnBelt < THIS^.cMAXBUFFERSIZE THEN
	m_intLastPaperIdx := (m_intLastPaperIdx + 1) MOD THIS^.cMAXBUFFERSIZE;
	m_arBuffer[m_intLastPaperIdx].udiItemId := In_udiItemId;
	m_arBuffer[m_intLastPaperIdx].lrePositionOnBelt_mm := 0.0;
	m_arBuffer[m_intLastPaperIdx].lrePositionOnBeltAdjusted_mm := 0.0;
	m_arBuffer[m_intLastPaperIdx].udiTimeOnBelt_us := 0;
	m_arBuffer[m_intLastPaperIdx].eStatus := E_PTR_Status.EnterBusy;
	m_intPaperOnBelt := m_intPaperOnBelt + 1;
	Push := TRUE;
END_IF
END_METHOD

METHOD PUBLIC Reset : BOOL
VAR_INPUT
END_VAR
m_intFirstPaperIdx := 0;
m_intLastPaperIdx := -1;
m_intPaperOnBelt := 0;
END_METHOD

PROPERTY PUBLIC TimeBase : UDINT
GET
TimeBase := m_udiTimeBase_us;
END_GET
SET
m_udiTimeBase_us := TimeBase;
END_SET
END_PROPERTY

END_FUNCTION_BLOCK

// POUs/Controller/Lvl1/MDC [Malteser Drive Controller]/FB_MDC
FUNCTION_BLOCK FB_MDC EXTENDS FB_CtrlBase
VAR_INPUT
	In_bolCrossPositionSensor			: BOOL;
	In_bolTablePositionSensor			: BOOL;
END_VAR
VAR_OUTPUT
	/// Position Output to the higher controller
	Out_intActualPosition				: INT;
END_VAR
VAR
	/// Specific interface struct for public access
	SIf					: T_Ctrl_SIf_MDC;
	///pointer to function block
	p_fbMotor			: POINTER TO FB_UMC;
	pMotor_CIF			: POINTER TO BASE_PLC.T_Ctrl_CIf;
END_VAR

(*__________________________________________________________________________________________________
¦	
¦	Vistaprint Schweiz GmbH
¦	CH - 8401 Winterthur
¦
¦	www.vistaprint.ch - info@vistaprint.ch
¦___________________________________________________________________________________________________

Function desription:
Vacuum Pump implementation. 


History:
Version		Date			Author		Comment
---------------------------------------------------------------------------------------------------
0.00.1		09.07.2013		PC			Start history
0.00.2		19.02.2014		AVME/MRU	Changes in sta_TurnBusy for simulation
0.00.3		24.02.2014		AVME/MRU	sta_OFFBusy reworked

___________________________________________________________________________________________________*)


IF (me.bolActivate) THEN // cyclic call enabled
	IF (CIf.Info.bolInitDone=FALSE) THEN // first cycle -> init
		CtrlInit();
		CIf.Info.bolInitDone := TRUE;
	ELSE
		CycleStartDuty();
	
		Always();
		
		StateMachine();
		
		CycleEndDuty();
	END_IF
END_IF;

PROPERTY ActualPosition : UINT
GET
ActualPosition := SIf.Cur.uintActualPosition;
END_GET
END_PROPERTY

METHOD PROTECTED Always : BOOL
SUPER^.Always();

// ----------------------------------------------------------------------------------
// cyclic actions outside of statemachine
IF (me.StateMachine.intState<>cSTA_SINGLE_ANSWER) THEN
	
	; // always error supervision
	
END_IF

// ----------------------------------------------------------------------------------
// Conditions Always
IF (((me.Alarm.eActivAlmClass=E_AlmClass.EOFF) OR (me.Alarm.eActivAlmClass=E_AlmClass.OFF) OR (me.intCmd=cCMD_OFF))
		 AND (me.StateMachine.intState<>cSTA_ERROR) AND (me.StateMachine.intState<>cSTA_ERRORQuit) AND
		(me.StateMachine.intState<>cSTA_OFF) AND (me.StateMachine.intState<>cSTA_OFFBusy)) THEN
	// alarm evt EOFF, OFF or cmd off
	me.StateMachine.intStateNext := cSTA_OFFBusy;
END_IF
END_METHOD

METHOD PROTECTED CtrlInit : BOOL
VAR_INPUT
END_VAR
SUPER^.CtrlInit();

// get child if
pMotor_CIF := AddChild(p_fbMotor^);
END_METHOD

PROPERTY PUBLIC CtrlSIf : POINTER TO T_Ctrl_SIf_MDC
GET
CtrlSIf := ADR(SIf);
END_GET
SET
END_SET
END_PROPERTY

PROPERTY PUBLIC Drive :  POINTER TO FB_UMC
GET
Drive := p_fbMotor;
END_GET
SET
p_fbMotor := Drive;
END_SET
END_PROPERTY

METHOD FB_init : BOOL
VAR_INPUT
	bInitRetains : BOOL; // if TRUE, the retain variables are initialized (warm start / cold start)
	bInCopyCode : BOOL;  // if TRUE, the instance afterwards gets moved into the copy code (online change)
END_VAR
VAR
	iIdx		: UINT;
	iLength		: UINT;	
END_VAR
//------------------------------------------------------------------------------------------------------------------------
// to manually change in new FUB implementation!!!
// define valid commands for this controller
iLength := SIZEOF(CIf.Job.aCmdList)/SIZEOF(CIf.Job.aCmdList[0]);
iIdx := 0;

WHILE (iIdx < iLength) AND (CIf.Job.aCmdList[iIdx].intCmd <> cCMD_INITIALIZED) DO
	iIdx := iIdx + 1; 
END_WHILE

IF (iIdx < iLength) THEN
// Add configuration of own comands	
	CIf.Job.aCmdList[iIdx].intCmd := MDC_CmdState.cCMD_INITIALIZE;
	CIf.Job.aCmdList[iIdx].strName := 'Initialize'; 
	CIf.Job.aCmdList[iIdx].bolAvailable := TRUE;
	iIdx := iIdx + 1;
	CIf.Job.aCmdList[iIdx].intCmd := MDC_CmdState.cCMD_TURN;
	CIf.Job.aCmdList[iIdx].strName := 'Turn'; 
	CIf.Job.aCmdList[iIdx].bolAvailable := TRUE;
	iIdx := iIdx + 1;
	CIf.Job.aCmdList[iIdx].intCmd := BASE_PLC.cCMD_RUN;
	CIf.Job.aCmdList[iIdx].strName := 'Run'; 
	CIf.Job.aCmdList[iIdx].bolAvailable := TRUE;
	iIdx := iIdx + 1;
	CIf.Job.aCmdList[iIdx].intCmd := MDC_CmdState.cCMD_PREPOSITION;
	CIf.Job.aCmdList[iIdx].strName := 'PrePosition'; 
	CIf.Job.aCmdList[iIdx].bolAvailable := TRUE;
	iIdx := iIdx + 1;
ELSE
	// Error if the aCmdList Array is to small
END_IF

// set name of class/typ
CIf.Info.strType := 'FB_MDC'; 

// set alarm class
SIf.Alm[E_ALM_MDC.TableSensorTimeout].eAlmClass := Base_PLC.E_AlmClass.TSTOP;
SIf.Alm[E_ALM_MDC.TableSensorTimeout].strText := 'Table Sensor Timeout'; 
SIf.Alm[E_ALM_MDC.CrossSensorTimeout].eAlmClass := Base_PLC.E_AlmClass.TSTOP;
SIf.Alm[E_ALM_MDC.CrossSensorTimeout].strText := 'Cross Sensor Timeout';
SIf.Alm[E_ALM_MDC.PositionSame].eAlmClass := Base_PLC.E_AlmClass.WARNING;
SIf.Alm[E_ALM_MDC.PositionSame].strText := 'New Position is the same as the actual position';

//*******************************************************************************
// initial values
//*******************************************************************************

// software configuration
CIf.SwCfg.bolExist := TRUE;
CIf.SwCfg.bolEnable := TRUE;
CIf.SwCfg.bolSimulation := FALSE;

// parameter
SIf.Cfg.uintPositionPerTurn			:= 4;
SIf.Par.intTurnDirection			:= 0;
SIf.Par.uinPositionToGo				:= 0;
SIf.Par.uinPositionSpeed_rpm		:= 1400;
SIf.Par.uinPrePositionSpeed_rpm		:= 450;
SIf.Par.udiInitializationTime_ms 	:= 16000;
SIf.Par.udiStepRotationTime_ms 		:= 2000;
SIf.Par.udiSimInitializationTime_ms := SIf.Par.udiInitializationTime_ms / 2;
SIf.Par.udiSimStepRotationTime_ms := SIf.Par.udiStepRotationTime_ms / 2;
SIf.Par.udiSimStartRotationTime_ms := SIf.Par.udiStepRotationTime_ms / 10;
END_METHOD

METHOD PROTECTED getCmdState : STRING

VAR_INPUT
	intCmdState: INT;
	bolState: BOOL;
END_VAR
getCmdState := SUPER^.getCmdState(intCmdState:=intCmdState,bolState:=bolState); // get global/base defined cmds/states

IF (getCmdState='') THEN // global not defined get local
	// get string cmd/state string information in runtime
	IF (bolState=FALSE) THEN
		CASE intCmdState OF
			MDC_CmdState.cCMD_INITIALIZE: 
				getCmdState := 'Initialize';
			MDC_CmdState.cCMD_TURN: 
				getCmdState := 'Turn';
			MDC_CmdState.cCMD_PREPOSITION: 
				getCmdState := 'PrePosition';
		END_CASE;
	ELSE
		// States's
		CASE intCmdState OF
			MDC_CmdState.cSTA_InitializeBusy: 
				getCmdState := 'InitializeBusy';
			MDC_CmdState.cSTA_InPositionBusy: 
				getCmdState := 'InPositionBusy';
			MDC_CmdState.cSTA_InPosition: 
				getCmdState := 'InPosition';
			MDC_CmdState.cSTA_StartTurnBusy: 
				getCmdState := 'StartTurnBusy';
			MDC_CmdState.cSTA_TurnBusy: 
				getCmdState := 'TurnBusy';
			MDC_CmdState.cSTA_TURNDONE: 
				getCmdState := 'TURNDONE';
			MDC_CmdState.cSTA_PREPOSITIONbusy: 
				getCmdState := 'PREPOSITIONbusy';
			MDC_CmdState.cSTA_PREPOSITION: 
				getCmdState := 'PREPOSITION';

			MDC_CmdState.cSUB_STOPbusy: 
				getCmdState := 'STOPbusy';
			MDC_CmdState.cSUB_TURNbusy: 
				getCmdState := 'TURNbusy';
			MDC_CmdState.cSUB_FINDHOLEbusy: 
				getCmdState := 'FINDHOLEbusy';
		END_CASE;
	END_IF
END_IF
END_METHOD

METHOD getCtrlSIf : POINTER TO T_Ctrl_SIf_MDC
getCtrlSIf := ADR(SIf);
END_METHOD

METHOD PROTECTED GetTurningDirection : E_TURN_DIRECTION
VAR
	iDifference 		: INT;
END_VAR
GetTurningDirection := E_TURN_DIRECTION.RIGHT;

// Determine the turning direction depending on set value or on shortest distance
CASE SIf.Par.intTurnDirection OF
	E_TURN_DIRECTION.LEFT	:
		GetTurningDirection := E_TURN_DIRECTION.LEFT;
	E_TURN_DIRECTION.AUTOMATIC 	:
		GetTurningDirection := E_TURN_DIRECTION.RIGHT;
		
		IF (SIf.Cur.uintActualPosition = 1) AND (SIf.Par.uinPositionToGo = 0) THEN
			iDifference := 0;
		END_IF

		iDifference := UINT_TO_INT(SIf.Par.uinPositionToGo - SIf.Cur.uintActualPosition);
		iDifference := ABS(iDifference);
		
		IF (    (SIf.Par.uinPositionToGo < SIf.Cur.uintActualPosition) AND (iDifference < UINT_TO_INT(SIf.Cfg.uintPositionPerTurn / 2)) 
			 OR (SIf.Par.uinPositionToGo > SIf.Cur.uintActualPosition) AND (iDifference > UINT_TO_INT(SIf.Cfg.uintPositionPerTurn / 2))) THEN
			GetTurningDirection := E_TURN_DIRECTION.LEFT;
		END_IF;
	E_TURN_DIRECTION.RIGHT	:
		GetTurningDirection := E_TURN_DIRECTION.RIGHT;
END_CASE;
END_METHOD

METHOD PROTECTED IncrementPosition : UINT
VAR_INPUT
	uinPosition		: UINT;
	eDirection		: E_TURN_DIRECTION;
END_VAR
VAR
	iNewPosition	: INT;
END_VAR
IF eDirection = E_TURN_DIRECTION.RIGHT THEN
	iNewPosition := UINT_TO_INT((uinPosition + 1) MOD SIf.Cfg.uintPositionPerTurn);
ELSE
	iNewPosition := UINT_TO_INT(uinPosition) - 1;
	
	IF (iNewPosition < 0) THEN
		iNewPosition := UINT_TO_INT(SIf.Cfg.uintPositionPerTurn) - 1;
	END_IF
END_IF

IncrementPosition := INT_TO_UINT(iNewPosition);
END_METHOD

METHOD PROTECTED IoInBridge : BOOL
// digitale and analoge inputs read from hardware or forcing
SIf.In.bolCrossPositionSensor.map := NOT THIS^.In_bolCrossPositionSensor;
SIf.In.bolTablePositionSensor.map := THIS^.In_bolTablePositionSensor;

IF (CIf.SwCfg.bolSimulation = FALSE) THEN
	getInBol(CIf.Job.bolIoForce,ADR(SIf.In.bolCrossPositionSensor));
	getInBol(CIf.Job.bolIoForce,ADR(SIf.In.bolTablePositionSensor));
ELSE
	//simulation of global IO
END_IF
END_METHOD

METHOD PROTECTED IoOutBridge : BOOL
VAR
	bolSwitchValvesOff: BOOL;
END_VAR
// digitale and analoge inputs read from hardware or forcing
IF (CIf.SwCfg.bolSimulation = FALSE) THEN
	setOutBol(CIf.Job.bolIoForce ,ADR(SIf.Out.intActualPosition));

	THIS^.Out_intActualPosition := SIf.Out.intActualPosition.map;
END_IF
END_METHOD

METHOD SetPositionToGo : BOOL
VAR_INPUT
	uinPositionToGo: UINT;
END_VAR
SIf.Par.uinPositionToGo := uinPositionToGo;

SetPositionToGo := uinPositionToGo = SIf.Cur.uintActualPosition;
END_METHOD

METHOD PROTECTED sta_ERROR : BOOL
// state implemetation
//--------------------------------------------------------------------------------------
// Entry action
	IF (me.StateMachine.intState<>me.StateMachine.intStateLastCycle) THEN
		me.StateMachine.intStateHistory := me.StateMachine.intStateLastCycle; // -> possibillity to go back to state before error
		me.StateMachine.intStateLastCycle := me.StateMachine.intState;
		pMotor_CIF^.Job.intACmd := BASE_PLC.cCMD_OFF;		
	END_IF


//--------------------------------------------------------------------------------------
// Cyclic action
	IF (me.StateMachine.intState=me.StateMachine.intStateLastCycle) THEN
		
		;
		
		
		// State Change Condition
		IF (CIf.Job.bolAlmReset = TRUE) THEN
			me.StateMachine.intStateNext := cSTA_ERRORQuit;
		END_IF
	END_IF




//--------------------------------------------------------------------------------------
// Exit action
	IF (me.StateMachine.intState<>me.StateMachine.intStateNext) THEN
		;
	END_IF
END_METHOD

METHOD PROTECTED sta_ERRORQuit : BOOL
// state implemetation
//--------------------------------------------------------------------------------------
// Entry action
	IF (me.StateMachine.intState<>me.StateMachine.intStateLastCycle) THEN
		me.StateMachine.intStateLastCycle := me.StateMachine.intState;
		
	END_IF


//--------------------------------------------------------------------------------------
// Cyclic action
	IF (me.StateMachine.intState=me.StateMachine.intStateLastCycle) THEN
		
		;
		// evtl. wait time if reset of device is necessary and then decide to go to states or ERROR state
		IF (CIf.Job.bolAlmReset = TRUE) THEN
			CIf.Job.eMe_ActivAlmClass := E_AlmClass.NONE; // reset feedback channel for parent
			CIf.Job.bolAlmReset := FALSE;
		END_IF
		
		// State Change Condition
		IF (CIf.Job.bolAlmReset = FALSE) THEN
			IF (me.StateMachine.intStateHistory<=cSTA_PON) THEN
				me.StateMachine.intStateNext := cSTA_PONBusy;
			ELSIF(me.intCmd=cCMD_OFF) THEN
				me.StateMachine.intStateNext := cSTA_OFFBusy;
			ELSIF(me.intCmd=cCMD_STOP) THEN
				me.StateMachine.intStateNext := cSTA_STOPBusy;
			ELSIF(me.intCmd=MDC_CmdState.cCMD_INITIALIZE) THEN
				me.StateMachine.intStateNext := MDC_CmdState.cSTA_InitializeBusy;
			ELSIF(me.intCmd=MDC_CmdState.cCMD_TURN) THEN
				me.StateMachine.intStateNext := MDC_CmdState.cSTA_InitializeBusy;
			END_IF
		END_IF
	END_IF




//--------------------------------------------------------------------------------------
// Exit action
	IF (me.StateMachine.intState<>me.StateMachine.intStateNext) THEN
		;
	END_IF
END_METHOD

METHOD PROTECTED sta_InitializeBusy : BOOL
VAR
	bCrossSensorPassed		: BOOL;
	bTableSensorPassed		: BOOL;
END_VAR
// state implemetation
//--------------------------------------------------------------------------------------
// Entry action
	IF (me.StateMachine.intState<>me.StateMachine.intStateLastCycle) THEN
		me.StateMachine.intStateLastCycle := me.StateMachine.intState;
		// Set Speed
		p_fbMotor^.CtrlSIf^.Par.uinSpeed_rpm := SIf.Par.uinPositionSpeed_rpm;
		pMotor_CIF^.Job.intACmd := UMC_CmdState.cCMD_RIGHT;		
		SIf.Cur.eActualTurningDirection := E_TURN_DIRECTION.RIGHT;

		fbSimulationTimer.IN := FALSE;
		fbSimulationTimer.PT := UDINT_TO_TIME(SIf.Par.udiSimInitializationTime_ms);
		fbSimulationTimer(); // set time/reset timer
		fbSimulationTimer.IN := TRUE; // start timer
		
		bCrossSensorPassed := FALSE;
		bTableSensorPassed := FALSE;
	END_IF


//--------------------------------------------------------------------------------------
// Cyclic action
	IF (me.StateMachine.intState=me.StateMachine.intStateLastCycle) THEN
		IF (CIf.SwCfg.bolSimulation) THEN
			fbSimulationTimer(); // simulation time

			IF (fbSimulationTimer.Q) THEN
				SIf.In.bolCrossPositionSensor.intern := TRUE;
				SIf.In.bolTablePositionSensor.intern := TRUE;				
			END_IF
		END_IF
		
		bCrossSensorPassed := bCrossSensorPassed OR SIf.In.bolCrossPositionSensor.intern;
		bTableSensorPassed := bTableSensorPassed OR SIf.In.bolTablePositionSensor.intern;
	
		IF (me.StateMachine.udiTimeInState_ms > SIf.Par.udiInitializationTime_ms) THEN
			IF NOT bCrossSensorPassed THEN
				pfbAlarmCtrl^.setAlarm(CIf.Info.intCtrlId,INT_TO_UINT(E_ALM_MDC.CrossSensorTimeout),0,ADR(SIf.Alm),E_AlmState.RST,CIf.Job.eMe_ActivAlmClass);
			END_IF
			
			IF NOT bTableSensorPassed THEN
				pfbAlarmCtrl^.setAlarm(CIf.Info.intCtrlId,INT_TO_UINT(E_ALM_MDC.TableSensorTimeout),0,ADR(SIf.Alm),E_AlmState.RST,CIf.Job.eMe_ActivAlmClass);
			END_IF
			
			me.StateMachine.intStateNext := Base_PLC.cSTA_ERROR;	
		END_IF

		IF SIf.In.bolCrossPositionSensor.intern AND SIf.In.bolTablePositionSensor.intern THEN
			me.StateMachine.intStateNext := MDC_CmdState.cSTA_InPositionBusy;
		END_IF
	END_IF


//--------------------------------------------------------------------------------------
// Exit action
	IF (me.StateMachine.intState<>me.StateMachine.intStateNext) THEN
		p_fbMotor^.CtrlSIf^.Par.uinSpeed_rpm := SIf.Par.uinPositionSpeed_rpm;
		SIf.Cur.uintActualPosition := 0;
	END_IF
END_METHOD

METHOD PROTECTED sta_InPosition : Bool
// state implemetation
//--------------------------------------------------------------------------------------
// Entry action
	IF (me.StateMachine.intState<>me.StateMachine.intStateLastCycle) THEN
		me.StateMachine.intStateLastCycle := me.StateMachine.intState;
		
		IF CIf.Job.intACmd = BASE_PLC.cCMD_RUN THEN
			CIf.Job.intACmd := cCMD_DONE;
		END_IF

		IF CIf.Job.intMCmd = BASE_PLC.cCMD_RUN THEN
			CIf.Job.intMCmd := cCMD_DONE;
		END_IF
	END_IF


//--------------------------------------------------------------------------------------
// Cyclic action
	IF (me.StateMachine.intState = me.StateMachine.intStateLastCycle) THEN
		CASE me.intCmd OF
			MDC_CmdState.cCMD_TURN,
			MDC_CmdState.cCMD_PREPOSITION:
//				IF SIf.Par.uinPositionToGo <> SIf.Cur.uintActualPosition THEN
//					SIf.Cur.eActualTurningDirection := GetTurningDirection();

					CASE me.intCmd OF
						MDC_CmdState.cCMD_TURN:
							me.StateMachine.intStateNext := MDC_CmdState.cSTA_StartTurnBusy;
						MDC_CmdState.cCMD_PREPOSITION:
							me.StateMachine.intStateNext := MDC_CmdState.cSTA_PREPOSITIONbusy;
					END_CASE
//				ELSE
//					CIf.Job.intACmd := cCMD_DONE;
//					CIf.Job.intMCmd := cCMD_DONE;
//					pfbAlarmCtrl^.setAlarm(CIf.Info.intCtrlId,INT_TO_UINT(E_ALM_MDC.PositionSame),0,ADR(SIf.Alm),E_AlmState.RST,CIf.Job.eMe_ActivAlmClass);
//				END_IF
				
			MDC_CmdState.cCMD_INITIALIZE:	
				me.StateMachine.intStateNext := MDC_CmdState.cSTA_InitializeBusy;
		END_CASE
	END_IF


//--------------------------------------------------------------------------------------
// Exit action
	IF (me.StateMachine.intState<>me.StateMachine.intStateNext) THEN
		;
	END_IF
END_METHOD

METHOD PROTECTED sta_InPositionBusy : BOOL
VAR_INPUT
END_VAR
// state implemetation
//--------------------------------------------------------------------------------------
// Entry action
	IF (me.StateMachine.intState<>me.StateMachine.intStateLastCycle) THEN
		me.StateMachine.intStateLastCycle := me.StateMachine.intState;
		pMotor_CIF^.Job.intACmd := BASE_PLC.cCMD_STOP;		
	END_IF


//--------------------------------------------------------------------------------------
// Cyclic action
	IF (me.StateMachine.intState=me.StateMachine.intStateLastCycle) THEN
		IF pMotor_CIF^.Job.intState = BASE_PLC.cSTA_STOP THEN
			me.StateMachine.intStateNext := MDC_CmdState.cSTA_InPosition;
		END_IF
	END_IF


//--------------------------------------------------------------------------------------
// Exit action
	IF (me.StateMachine.intState<>me.StateMachine.intStateNext) THEN
		;
	END_IF
END_METHOD

METHOD PROTECTED sta_OFF : BOOL
VAR_INPUT
END_VAR
// state implemetation
//--------------------------------------------------------------------------------------
// Entry action
	IF (me.StateMachine.intState<>me.StateMachine.intStateLastCycle) THEN
		me.StateMachine.intStateLastCycle := me.StateMachine.intState;

	END_IF


//--------------------------------------------------------------------------------------
// Cyclic action
	IF (me.StateMachine.intState=me.StateMachine.intStateLastCycle) THEN
		IF me.intCmd = MDC_CmdState.cCMD_INITIALIZE THEN
			me.StateMachine.intStateNext := MDC_CmdState.cSTA_InitializeBusy;
		END_IF
	END_IF


//--------------------------------------------------------------------------------------
// Exit action
	IF (me.StateMachine.intState<>me.StateMachine.intStateNext) THEN
		;
	END_IF
END_METHOD

METHOD PROTECTED sta_OFFBusy : BOOL
VAR_INPUT
END_VAR
// state implemetation
//--------------------------------------------------------------------------------------
// Entry action
	IF (me.StateMachine.intState<>me.StateMachine.intStateLastCycle) THEN
		me.StateMachine.intStateLastCycle := me.StateMachine.intState;
		pMotor_CIF^.Job.intACmd := BASE_PLC.cCMD_OFF;		
	END_IF


//--------------------------------------------------------------------------------------
// Cyclic action
	IF (me.StateMachine.intState=me.StateMachine.intStateLastCycle) THEN
		// Set commandos not only in entry action because of possible errors or manual/auto changes
		pMotor_CIF^.Job.intACmd := BASE_PLC.cCMD_OFF;		

		IF pMotor_CIF^.Job.intState = BASE_PLC.cSTA_OFF THEN
			me.StateMachine.intStateNext := BASE_PLC.cSTA_OFF;
		END_IF
	END_IF


//--------------------------------------------------------------------------------------
// Exit action
	IF (me.StateMachine.intState<>me.StateMachine.intStateNext) THEN
		;
	END_IF
END_METHOD

METHOD PROTECTED sta_PON : BOOL
VAR_INPUT
END_VAR
// state implemetation
//--------------------------------------------------------------------------------------
// Entry action
	IF (me.StateMachine.intState<>me.StateMachine.intStateLastCycle) THEN
		me.StateMachine.intStateLastCycle := me.StateMachine.intState;
		
	END_IF


//--------------------------------------------------------------------------------------
// Cyclic action
	IF (me.StateMachine.intState=me.StateMachine.intStateLastCycle) THEN
		;
	END_IF




//--------------------------------------------------------------------------------------
// Exit action
	IF (me.StateMachine.intState<>me.StateMachine.intStateNext) THEN
		;
	END_IF
END_METHOD

METHOD PROTECTED sta_PREPOSITION : BOOL
VAR_INPUT
END_VAR
// state implemetation
//--------------------------------------------------------------------------------------
// Entry action
IF (me.StateMachine.intState<>me.StateMachine.intStateLastCycle) THEN
	me.StateMachine.intStateLastCycle := me.StateMachine.intState;

	CIf.Job.intACmd := cCMD_DONE;
	CIf.Job.intMCmd := cCMD_DONE;
END_IF


//--------------------------------------------------------------------------------------
// Cyclic action
IF (me.StateMachine.intState=me.StateMachine.intStateLastCycle) THEN
	CASE me.intCmd OF
		MDC_CmdState.cCMD_INITIALIZE:
			me.StateMachine.intStateNext := MDC_CmdState.cSTA_InitializeBusy;
		MDC_CmdState.cCMD_TURN:
			me.StateMachine.intStateNext := MDC_CmdState.cSTA_StartTurnBusy;
		BASE_PLC.cCMD_RUN:
			me.StateMachine.intStateNext := MDC_CmdState.cSTA_InPositionBusy;
	END_CASE
END_IF


//--------------------------------------------------------------------------------------
// Exit action
IF (me.StateMachine.intState<>me.StateMachine.intStateNext) THEN
	;
END_IF
END_METHOD

METHOD PROTECTED sta_PREPOSITIONbusy : BOOL
VAR_INPUT
END_VAR
VAR
	eOldDirection		: BASE_ELEMENTS.E_TURN_DIRECTION;
END_VAR
// state implemetation
//--------------------------------------------------------------------------------------
// Entry action
IF (me.StateMachine.intState<>me.StateMachine.intStateLastCycle) THEN
	me.StateMachine.intStateLastCycle := me.StateMachine.intState;
	
	IF SIf.Par.uinPositionToGo <> SIf.Cur.uintActualPosition THEN
		eOldDirection := SIf.Cur.eActualTurningDirection;
		SIf.Cur.eActualTurningDirection := GetTurningDirection();

		// Set Speed
		p_fbMotor^.CtrlSIf^.Par.uinSpeed_rpm := SIf.Par.uinPrePositionSpeed_rpm;
		
		// Send the comand
		CASE SIf.Cur.eActualTurningDirection OF
			E_TURN_DIRECTION.LEFT:
				pMotor_CIF^.Job.intACmd := cCMD_LEFT;		
			E_TURN_DIRECTION.RIGHT:
				pMotor_CIF^.Job.intACmd := cCMD_RIGHT;		
		END_CASE

		fbSimulationTimer.IN := FALSE;
		fbSimulationTimer.PT := UDINT_TO_TIME(SIf.Par.udiSimStartRotationTime_ms);
		fbSimulationTimer(); // set time/reset timer
		fbSimulationTimer.IN := TRUE; // start timer
		
		IF eOldDirection = SIf.Cur.eActualTurningDirection THEN
			me.SubStateMachine.intState	    := MDC_CmdState.cSUB_TURNbusy;
			me.SubStateMachine.intStateNext := MDC_CmdState.cSUB_TURNbusy;
		ELSE
			me.SubStateMachine.intState	    := MDC_CmdState.cSUB_FINDHOLEbusy;
			me.SubStateMachine.intStateNext := MDC_CmdState.cSUB_FINDHOLEbusy;
		END_IF
	ELSE
		me.StateMachine.intStateNext := MDC_CmdState.cSTA_PREPOSITION;
	END_IF
END_IF


//--------------------------------------------------------------------------------------
// Cyclic action
IF (me.StateMachine.intState=me.StateMachine.intStateLastCycle) THEN
	IF (CIf.SwCfg.bolSimulation) THEN
		fbSimulationTimer(); // simulation time

		IF (fbSimulationTimer.Q) THEN
			SIf.In.bolCrossPositionSensor.intern := FALSE;
			SIf.In.bolTablePositionSensor.intern := FALSE;
		END_IF
	END_IF
	
	CASE me.SubStateMachine.intState OF
		MDC_CmdState.cSUB_FINDHOLEbusy:
			IF SIf.In.bolCrossPositionSensor.intern THEN
				me.SubStateMachine.intStateNext := MDC_CmdState.cSUB_TURNbusy;
			END_IF
		MDC_CmdState.cSUB_TURNbusy:
			IF NOT SIf.In.bolCrossPositionSensor.intern THEN
				pMotor_CIF^.Job.intACmd := BASE_PLC.cCMD_STOP;		
				me.SubStateMachine.intStateNext := MDC_CmdState.cSUB_STOPbusy;
			END_IF
		MDC_CmdState.cSUB_STOPbusy:
			IF pMotor_CIF^.Job.intState = BASE_PLC.cSTA_STOP THEN
				me.StateMachine.intStateNext := MDC_CmdState.cSTA_PREPOSITION;
			END_IF
	END_CASE
	
	IF me.intCmd = MDC_CmdState.cCMD_TURN THEN
//		Log Message ---------------------
		TC2_SYSTEM.ADSLOGSTR(ADSLOG_MSGTYPE_LOG,'sta_PREPOSITIONbusy, %s','MDC_CmdState.cCMD_TURN');
//		---------------------------------
		
		IF SIf.Par.uinPositionToGo <> SIf.Cur.uintActualPosition THEN
			me.StateMachine.intStateNext := MDC_CmdState.cSTA_StartTurnBusy;
		ELSE
			CIf.Job.intACmd := cCMD_DONE;
			CIf.Job.intMCmd := cCMD_DONE;
			pfbAlarmCtrl^.setAlarm(CIf.Info.intCtrlId,INT_TO_UINT(E_ALM_MDC.PositionSame),0,ADR(SIf.Alm),E_AlmState.RST,CIf.Job.eMe_ActivAlmClass);
		END_IF
	END_IF

	IF (me.StateMachine.udiTimeInState_ms > SIf.Par.udiStepRotationTime_ms) THEN
		pfbAlarmCtrl^.setAlarm(CIf.Info.intCtrlId,INT_TO_UINT(E_ALM_MDC.CrossSensorTimeout),0,ADR(SIf.Alm),E_AlmState.RST,CIf.Job.eMe_ActivAlmClass);
		me.StateMachine.intStateNext := Base_PLC.cSTA_ERROR;	
	END_IF
	
	
END_IF


//--------------------------------------------------------------------------------------
// Exit action
IF (me.StateMachine.intState<>me.StateMachine.intStateNext) THEN
	;
END_IF
END_METHOD

METHOD PROTECTED sta_StartTurnBusy : Bool
VAR
	iDifference			: INT;
	eOldDirection		: BASE_ELEMENTS.E_TURN_DIRECTION;
END_VAR
// state implemetation
//--------------------------------------------------------------------------------------
// Entry action
	IF (me.StateMachine.intState<>me.StateMachine.intStateLastCycle) THEN
		me.StateMachine.intStateLastCycle := me.StateMachine.intState;
		
		IF SIf.Par.uinPositionToGo <> SIf.Cur.uintActualPosition THEN
			eOldDirection := SIf.Cur.eActualTurningDirection;
			SIf.Cur.eActualTurningDirection := GetTurningDirection();

			// Set Speed
			p_fbMotor^.CtrlSIf^.Par.uinSpeed_rpm := SIf.Par.uinPositionSpeed_rpm;
			
			// Send the comand
			CASE SIf.Cur.eActualTurningDirection OF
				E_TURN_DIRECTION.LEFT:
					pMotor_CIF^.Job.intACmd := cCMD_LEFT;		
				E_TURN_DIRECTION.RIGHT:
					pMotor_CIF^.Job.intACmd := cCMD_RIGHT;		
			END_CASE

			IF eOldDirection = SIf.Cur.eActualTurningDirection THEN
				me.SubStateMachine.intState	    := MDC_CmdState.cSUB_TURNbusy;
				me.SubStateMachine.intStateNext := MDC_CmdState.cSUB_TURNbusy;
			ELSE
				me.SubStateMachine.intState	    := MDC_CmdState.cSUB_FINDHOLEbusy;
				me.SubStateMachine.intStateNext := MDC_CmdState.cSUB_FINDHOLEbusy;
			END_IF
			
			fbSimulationTimer.IN := FALSE;
			fbSimulationTimer.PT := UDINT_TO_TIME(SIf.Par.udiSimStartRotationTime_ms);
			fbSimulationTimer(); // set time/reset timer
			fbSimulationTimer.IN := TRUE; // start timer
		END_IF
	END_IF


//--------------------------------------------------------------------------------------
// Cyclic action
	IF (me.StateMachine.intState=me.StateMachine.intStateLastCycle) THEN
		IF (CIf.SwCfg.bolSimulation) THEN
			fbSimulationTimer(); // simulation time

			IF (fbSimulationTimer.Q) THEN
				SIf.In.bolCrossPositionSensor.intern := FALSE;
				SIf.In.bolTablePositionSensor.intern := FALSE;
			END_IF
		END_IF
		
		CASE me.SubStateMachine.intState OF
			MDC_CmdState.cSUB_FINDHOLEbusy:
				IF SIf.In.bolCrossPositionSensor.intern THEN
					me.SubStateMachine.intStateNext := MDC_CmdState.cSUB_TURNbusy;
				END_IF
			MDC_CmdState.cSUB_TURNbusy:
				IF NOT SIf.In.bolCrossPositionSensor.intern THEN
					me.StateMachine.intStateNext := MDC_CmdState.cSTA_TurnBusy;
				END_IF
		END_CASE

		IF SIf.Par.uinPositionToGo = SIf.Cur.uintActualPosition THEN
			me.StateMachine.intStateNext := MDC_CmdState.cSTA_TURNDONE;
		END_IF 
		
		IF (me.StateMachine.udiTimeInState_ms > SIf.Par.udiStepRotationTime_ms) THEN
			pfbAlarmCtrl^.setAlarm(CIf.Info.intCtrlId,INT_TO_UINT(E_ALM_MDC.CrossSensorTimeout),0,ADR(SIf.Alm),E_AlmState.RST,CIf.Job.eMe_ActivAlmClass);
			me.StateMachine.intStateNext := Base_PLC.cSTA_ERROR;	
		END_IF
	END_IF


//--------------------------------------------------------------------------------------
// Exit action
	IF (me.StateMachine.intState<>me.StateMachine.intStateNext) THEN
		;
	END_IF
END_METHOD

METHOD PROTECTED sta_TurnBusy : Bool
VAR_INPUT
END_VAR
// state implemetation
//--------------------------------------------------------------------------------------
// Entry action
	IF (me.StateMachine.intState<>me.StateMachine.intStateLastCycle) THEN
		me.StateMachine.intStateLastCycle := me.StateMachine.intState;

		fbSimulationTimer.IN := FALSE;
		fbSimulationTimer.PT := UDINT_TO_TIME(SIf.Par.udiSimStepRotationTime_ms);
		fbSimulationTimer(); // set time/reset timer
		fbSimulationTimer.IN := TRUE; // start timer

		me.SubStateMachine.intState 	:= MDC_CmdState.cSUB_TURNbusy;
		me.SubStateMachine.intStateNext := MDC_CmdState.cSUB_TURNbusy;
	END_IF


//--------------------------------------------------------------------------------------
// Cyclic action
	IF (me.StateMachine.intState=me.StateMachine.intStateLastCycle) THEN
		IF (CIf.SwCfg.bolSimulation) THEN
			fbSimulationTimer(); // simulation time

			IF (fbSimulationTimer.Q) THEN
				SIf.In.bolCrossPositionSensor.intern := TRUE;
			END_IF
		END_IF
		
		CASE me.SubStateMachine.intState OF
			MDC_CmdState.cSUB_TURNbusy:
				IF SIf.In.bolCrossPositionSensor.intern THEN
					SIf.Cur.uintActualPosition := IncrementPosition(SIf.Cur.uintActualPosition,SIf.Cur.eActualTurningDirection);
					
					IF (CIf.SwCfg.bolSimulation) THEN
						IF SIf.Cur.uintActualPosition = 0 THEN
							SIf.In.bolTablePositionSensor.intern := TRUE;
						END_IF
					END_IF
					
					IF SIf.Par.uinPositionToGo = SIf.Cur.uintActualPosition THEN
						pMotor_CIF^.Job.intACmd := BASE_PLC.cCMD_STOP;		
						me.SubStateMachine.intStateNext := MDC_CmdState.cSUB_STOPbusy;
					ELSE
						me.StateMachine.intStateNext := MDC_CmdState.cSTA_StartTurnBusy;
					END_IF 
				END_IF
				
			MDC_CmdState.cSUB_STOPbusy:
				IF pMotor_CIF^.Job.intState = BASE_PLC.cSTA_STOP THEN
					me.StateMachine.intStateNext := MDC_CmdState.cSTA_TURNDONE;
				END_IF
		END_CASE


		IF (me.StateMachine.udiTimeInState_ms > SIf.Par.udiStepRotationTime_ms) THEN
			pfbAlarmCtrl^.setAlarm(CIf.Info.intCtrlId,INT_TO_UINT(E_ALM_MDC.CrossSensorTimeout),0,ADR(SIf.Alm),E_AlmState.RST,CIf.Job.eMe_ActivAlmClass);
			me.StateMachine.intStateNext := Base_PLC.cSTA_ERROR;	
		END_IF
	END_IF


//--------------------------------------------------------------------------------------
// Exit action
	IF (me.StateMachine.intState<>me.StateMachine.intStateNext) THEN
		;
	END_IF
END_METHOD

METHOD PROTECTED sta_TURNDONE : BOOL
VAR_INPUT
END_VAR
// state implemetation
//--------------------------------------------------------------------------------------
// Entry action
IF (me.StateMachine.intState<>me.StateMachine.intStateLastCycle) THEN
	me.StateMachine.intStateLastCycle := me.StateMachine.intState;
	
	IF CIf.Job.intACmd = MDC_CmdState.cCMD_TURN THEN
		CIf.Job.intACmd := cCMD_DONE;
	END_IF
	
	IF CIf.Job.intMCmd = MDC_CmdState.cCMD_TURN THEN
		CIf.Job.intMCmd := cCMD_DONE;
	END_IF
END_IF


//--------------------------------------------------------------------------------------
// Cyclic action
IF (me.StateMachine.intState=me.StateMachine.intStateLastCycle) THEN
	CASE me.intCmd OF
		MDC_CmdState.cCMD_INITIALIZE:
			me.StateMachine.intStateNext := MDC_CmdState.cSTA_InitializeBusy;
		BASE_PLC.cCMD_RUN:
			me.StateMachine.intStateNext := MDC_CmdState.cSTA_InPositionBusy;
	END_CASE
END_IF


//--------------------------------------------------------------------------------------
// Exit action
IF (me.StateMachine.intState<>me.StateMachine.intStateNext) THEN
	;
END_IF
END_METHOD

METHOD PROTECTED StateMachine : BOOL
SUPER^.StateMachine();

// main statemachine of base controller
CASE me.StateMachine.intState OF
    MDC_CmdState.cSTA_InitializeBusy: 
        THIS^.sta_InitializeBusy();
    MDC_CmdState.cSTA_InPositionBusy: 
        THIS^.sta_InPositionBusy();
    MDC_CmdState.cSTA_InPosition: 
        THIS^.sta_InPosition();
    MDC_CmdState.cSTA_StartTurnBusy: 
        THIS^.sta_StartTurnBusy();
    MDC_CmdState.cSTA_TurnBusy: 
        THIS^.sta_TurnBusy();
    MDC_CmdState.cSTA_PREPOSITION: 
        THIS^.sta_PREPOSITION();
    MDC_CmdState.cSTA_PREPOSITIONbusy: 
        THIS^.sta_PREPOSITIONbusy();
    MDC_CmdState.cSTA_TURNDONE: 
        THIS^.sta_TURNDONE();
END_CASE;
END_METHOD

END_FUNCTION_BLOCK

// POUs/Controller/Lvl1/PTB [Paper Transport Belt]/FB_PTB
FUNCTION_BLOCK FB_PTB EXTENDS FB_CtrlBase
VAR_INPUT
	In_bolBeltEntrySensor		: BOOL;
	In_bolBeltExitSensor		: BOOL;
END_VAR
VAR_OUTPUT
END_VAR
VAR
	/// Specific interface struct for public access
	SIf					: T_Ctrl_SIf_PTB;
	///pointer to function block
	p_fbMotor				: POINTER TO FB_UMC;
	pMotorCIf				: POINTER TO T_Ctrl_CIf;
	p_fbPump				: POINTER TO FB_VPC;
	pPumpCIf				: POINTER TO T_Ctrl_CIf;
	fbEntrySensorDebounce	: FB_PRS;
	fbExitSensorDebounce	: FB_PRS;
	arMotorDirection		: ARRAY [0..E_BELT_DIRECTION.MAX_E_BELT_DIRECTION-1] OF E_TURN_DIRECTION;
	
	// Paper Position Service
	fbPositionService		: FB_PTR;
	udiIdCounter			: UDINT;
	
	// Paper Edge Detectors
	fbPaperEntryPEdge					: TC2_STANDARD.R_TRIG;
	fbPaperEntryNEdge					: TC2_STANDARD.F_TRIG;
	fbPaperExitPEdge					: TC2_STANDARD.R_TRIG;
	fbPaperExitNEdge					: TC2_STANDARD.F_TRIG;
	
END_VAR

(*__________________________________________________________________________________________________
¦	
¦	Vistaprint Schweiz GmbH
¦	CH - 8401 Winterthur
¦
¦	www.vistaprint.ch - info@vistaprint.ch
¦___________________________________________________________________________________________________

Function desription:
Vacuum Pump implementation. 


History:
Version		Date			Author		Comment
---------------------------------------------------------------------------------------------------
0.00.1		09.07.2013		PC			Start history
0.00.2		14.02.2014		AVME/MRU	Cyclic call of fbPositionService added
0.00.3		24.02.2014		AVME/MRU	sta_OFFBusy reworked
___________________________________________________________________________________________________*)


IF (me.bolActivate) THEN // cyclic call enabled
	IF (CIf.Info.bolInitDone=FALSE) THEN // first cycle -> init
		CtrlInit();
		CIf.Info.bolInitDone := TRUE;
	ELSE
		CycleStartDuty();
	
		Always();
		
		StateMachine();
		
		CycleEndDuty();
	END_IF
END_IF;

METHOD PROTECTED Always : BOOL
SUPER^.Always();

// ----------------------------------------------------------------------------------
// cyclic actions outside of statemachine
IF (me.StateMachine.intState<>cSTA_SINGLE_ANSWER) THEN
	
	; // always error supervision
	
END_IF

// ----------------------------------------------------------------------------------
// Conditions Always
IF (((me.Alarm.eActivAlmClass=E_AlmClass.EOFF) OR (me.Alarm.eActivAlmClass=E_AlmClass.OFF) OR (me.intCmd=cCMD_OFF))
		 AND (me.StateMachine.intState<>cSTA_ERROR) AND (me.StateMachine.intState<>cSTA_ERRORQuit) AND
		(me.StateMachine.intState<>cSTA_OFF) AND (me.StateMachine.intState<>cSTA_OFFBusy)) THEN
	// alarm evt EOFF, OFF or cmd off
	me.StateMachine.intStateNext := cSTA_OFFBusy;
END_IF

// ----------------------------------------------------------------------------------
// Conditions Always
// overrule error always from base -> no EOFF State!! in EOFF go to OFF
IF (me.StateMachine.intStateNext = cSTA_EOFFBusy) THEN
	IF (me.StateMachine.intState=cSTA_OFF) THEN
		me.StateMachine.intStateNext := cSTA_OFF;
	ELSE // stay in OFF
		me.StateMachine.intStateNext := cSTA_OFFBusy;
	END_IF
END_IF

// -----------------------------------------------------------------------------------
PaperPositionHandling();
// -----------------------------------------------------------------------------------
END_METHOD

METHOD PROTECTED CalculateBeltParameter : UINT
VAR_INPUT
	uinBeltSpeed_mms		: UINT;   	// Belt speed in mm/sec
	reaRpmDistance			: REAL;		// mm/rotation
	pCur		: POINTER TO T_Belt_Cur_Base;
END_VAR
pCur^.uinBeltSpeed_mms := uinBeltSpeed_mms;
// RPM = Speed [mm/sec] / Dispance per Rotation [mm/rpm]
pCur^.uinBeltSpeed_rpm := REAL_TO_UINT(UINT_TO_REAL(uinBeltSpeed_mms) * 60.0 / reaRpmDistance);

CalculateBeltParameter := pCur^.uinBeltSpeed_rpm;
END_METHOD

METHOD PROTECTED CalculateModeParameter : BOOL
VAR_INPUT
END_VAR
CASE SIf.Cfg.eMode OF  
	E_PTB_MODE.ToDistance:
		SIf.Cur.udiTimeToMove_ms		:= REAL_TO_UDINT( 1000.0 * UDINT_TO_REAL(SIf.Par.udiDistanceToMove_mm) / UINT_TO_REAL(SIf.Par.rBeltParam.uinBeltSpeed));
		SIf.Cur.udiTimeToMove_ms		:= SIf.Cur.udiTimeToMove_ms + p_fbMotor^.CtrlSIf^.Par.udiMoveStartLatency - p_fbMotor^.CtrlSIf^.Par.udiMoveStopLatency;
		SIf.Cur.udiDistanceToMove_mm	:= SIf.Par.udiDistanceToMove_mm;
	E_PTB_MODE.ToTime:
		SIf.Cur.udiTimeToMove_ms		:= SIf.Par.udiTimeToMove_ms;
		SIf.Cur.udiDistanceToMove_mm	:= SIf.Par.udiTimeToMove_ms * UINT_TO_UDINT(SIf.Par.rBeltParam.uinBeltSpeed) / 1000;
		SIf.Cur.udiTimeToMove_ms		:= SIf.Cur.udiTimeToMove_ms + p_fbMotor^.CtrlSIf^.Par.udiMoveStartLatency - p_fbMotor^.CtrlSIf^.Par.udiMoveStopLatency;
ELSE
	SIf.Cur.udiTimeToMove_ms		:= 0;
	SIf.Cur.udiDistanceToMove_mm	:= 0;
END_CASE
END_METHOD

METHOD PROTECTED CheckPumpState : BOOL
VAR_INPUT
	intState		: INT;
END_VAR
CheckPumpState := TRUE;

IF SIf.Cfg.bolVacuumPresent THEN
	CheckPumpState := p_fbPump^.CtrlCIf^.Job.intState = intState;
END_IF
END_METHOD

ACTION cmd_OFF:
p_fbMotor^.CtrlCIf^.Job.intACmd := BASE_PLC.cCMD_OFF;
SetPumpComand(cCMD_OFF);
END_ACTION

METHOD PROTECTED cmd_RUN : BOOL
VAR_INPUT
	uinBeltSpeed			: UINT;
END_VAR
SIf.Cur.eActualDirection := SIf.Par.intDirection;
SIf.Cur.rBeltParam.uinBeltSpeed_rpm := CalculateBeltParameter(
											uinBeltSpeed,
											sif.Cfg.rBeltParam.reaRpmDistance_mm,
											ADR(SIf.Cur.rBeltParam));
CalculateModeParameter();
p_fbMotor^.CtrlSIf^.Par.eRotationDirection 	:= THIS^.arMotorDirection[SIf.Par.intDirection];
p_fbMotor^.CtrlSIf^.Par.uinSpeed_rpm 		:= SIf.Cur.rBeltParam.uinBeltSpeed_rpm;
p_fbMotor^.CtrlCIf^.Job.intACmd :=BASE_PLC.cCMD_RUN;
SetPumpComand(cCMD_RUN);
END_METHOD

ACTION cmd_STOP:
p_fbMotor^.CtrlCIf^.Job.intACmd := BASE_PLC.cCMD_STOP;
SetPumpComand(cCMD_RUN);
END_ACTION

METHOD PROTECTED CtrlInit : BOOL
VAR_INPUT
END_VAR
SUPER^.CtrlInit();

pMotorCIf := p_fbMotor^.CtrlCIf;
AddChild(p_fbMotor^);

IF SIf.Cfg.bolVacuumPresent THEN
	pPumpCIf  := p_fbPump^.CtrlCIf;
	AddChild(p_fbPump^);
END_IF

arMotorDirection[E_BELT_DIRECTION.BACKWARD] := SIf.Cfg.rBeltParam.intBackwardDirection;
arMotorDirection[E_BELT_DIRECTION.FORWARD] := SIf.Cfg.rBeltParam.intForwardDirection;

fbPositionService.TimeBase := me.FUBInfo.udiSample_us;
fbPositionService.BeltLength := UDINT_TO_DINT(SIf.Par.udiBeltLength_mm);

CASE SIf.Par.ePaperOrientation OF
	E_PTB_PaperDirection.Portrait:
		fbPositionService.PaperEntryOffset := UINT_TO_INT(SIf.Par.uinPaperHight_mm); 
	E_PTB_PaperDirection.Landscape:
		fbPositionService.PaperEntryOffset := UINT_TO_INT(SIf.Par.uinPaperWidth_mm); 
END_CASE

SIf.Cur.pPositionList := fbPositionService.PositionList;
udiIdCounter := 0;
END_METHOD

PROPERTY PUBLIC CtrlSIf : POINTER TO T_Ctrl_SIf_PTB
GET
CtrlSIf := ADR(SIf);
END_GET
SET
END_SET
END_PROPERTY

PROPERTY PUBLIC Drive :  POINTER TO FB_UMC
GET
Drive := p_fbMotor;
END_GET
SET
p_fbMotor := Drive;
END_SET
END_PROPERTY

METHOD FB_init : BOOL
VAR_INPUT
	bInitRetains : BOOL; // if TRUE, the retain variables are initialized (warm start / cold start)
	bInCopyCode : BOOL;  // if TRUE, the instance afterwards gets moved into the copy code (online change)
END_VAR
VAR
	iIdx		: UINT;
	iLength		: UINT;	
END_VAR
//------------------------------------------------------------------------------------------------------------------------
// to manually change in new FUB implementation!!!
// define valid commands for this controller
iLength := SIZEOF(CIf.Job.aCmdList)/SIZEOF(CIf.Job.aCmdList[0]);
iIdx := 0;

WHILE (iIdx < iLength) AND (CIf.Job.aCmdList[iIdx].intCmd <> cCMD_INITIALIZED) DO
	iIdx := iIdx + 1; 
END_WHILE

IF (iIdx < iLength) THEN
// Add configuration of own comands	
	CIf.Job.aCmdList[iIdx].intCmd := BASE_PLC.cCMD_RUN;
	CIf.Job.aCmdList[iIdx].strName := 'Run'; 
	CIf.Job.aCmdList[iIdx].bolAvailable := TRUE;
	iIdx := iIdx + 1;
	CIf.Job.aCmdList[iIdx].intCmd := BASE_PLC.cCMD_STOP;
	CIf.Job.aCmdList[iIdx].strName := 'Stop'; 
	CIf.Job.aCmdList[iIdx].bolAvailable := TRUE;
	iIdx := iIdx + 1;
	CIf.Job.aCmdList[iIdx].intCmd := PTB_CmdState.cCMD_EJECTPAPER;
	CIf.Job.aCmdList[iIdx].strName := 'EJECTPAPER'; 
	CIf.Job.aCmdList[iIdx].bolAvailable := TRUE;
	iIdx := iIdx + 1;
	CIf.Job.aCmdList[iIdx].intCmd := PTB_CmdState.cCMD_STACKPAPER;
	CIf.Job.aCmdList[iIdx].strName := 'STACKPAPER'; 
	CIf.Job.aCmdList[iIdx].bolAvailable := TRUE;
ELSE
	// Error if the aCmdList Array is to small
END_IF

// set name of class/typ
CIf.Info.strType := 'FB_PTB'; 

// set alarm class

SIf.Alm[E_ALM_PTB.TestAlarm].eAlmClass := Base_PLC.E_AlmClass.TSTOP;
SIf.Alm[E_ALM_PTB.TestAlarm].strText := 'Baum' ;


//*******************************************************************************
// initial values
//*******************************************************************************

// software configuration
CIf.SwCfg.bolExist := TRUE;
CIf.SwCfg.bolEnable := TRUE;
CIf.SwCfg.bolSimulation := FALSE;

// configuration
SIf.Cfg.rBeltParam.intBackwardDirection		:= E_TURN_DIRECTION.LEFT;
SIf.Cfg.rBeltParam.intForwardDirection		:= E_TURN_DIRECTION.RIGHT;
SIf.Cfg.bolVacuumPresent					:= TRUE;
SIf.Cfg.eMode								:= E_PTB_MODE.Endless;
SIf.Cfg.rBeltParam.reaRpmDistance_mm		:= 20.3;

// parameter
SIf.Par.intDirection				:= E_BELT_DIRECTION.FORWARD;
SIf.Par.rBeltParam.uinBeltSpeed		:= 412;
SIf.Par.udiDistanceToMove_mm		:= 0;
SIf.Par.udiTimeToMove_ms			:= 0;
SIf.Par.ePaperOrientation			:= E_PTB_PaperDirection.Portrait;
SIf.Par.uinPaperHight_mm			:= 460;
SIf.Par.uinPaperWidth_mm			:= 320;
SIf.Par.uinInputSignalDebounceTime_ms := 50;


fbEntrySensorDebounce.CtrlSIf^.Par.udiDebounceAbsentTime_ms := SIf.Par.uinInputSignalDebounceTime_ms;
fbEntrySensorDebounce.CtrlSIf^.Par.udiDebouncePresentTime_ms := SIf.Par.uinInputSignalDebounceTime_ms;
fbExitSensorDebounce.CtrlSIf^.Par.udiDebounceAbsentTime_ms := SIf.Par.uinInputSignalDebounceTime_ms;
fbExitSensorDebounce.CtrlSIf^.Par.udiDebouncePresentTime_ms := SIf.Par.uinInputSignalDebounceTime_ms;
END_METHOD

METHOD PROTECTED getCmdState : STRING

VAR_INPUT
	intCmdState: INT;
	bolState: BOOL;
END_VAR
getCmdState := SUPER^.getCmdState(intCmdState:=intCmdState,bolState:=bolState); // get global/base defined cmds/states

IF (getCmdState='') THEN // global not defined get local
	// get string cmd/state string information in runtime
	IF (bolState=FALSE) THEN
		CASE intCmdState OF
			PTB_CmdState.cCMD_EJECTPAPER: 
				getCmdState := 'EJECTPAPER';
			PTB_CmdState.cCMD_STACKPAPER: 
				getCmdState := 'STACKPAPER';
		END_CASE;
	ELSE
		// States's
		CASE intCmdState OF
			PTB_CmdState.cSTA_EJECTPAPER: 
				getCmdState := 'EJECTPAPER';
			PTB_CmdState.cSTA_EJECTPAPERbusy: 
				getCmdState := 'EJECTPAPERbusy';
			PTB_CmdState.cSTA_STACKPAPER: 
				getCmdState := 'STACKPAPER';
			PTB_CmdState.cSTA_STACKPAPERbusy: 
				getCmdState := 'STACKPAPERbusy';
			PTB_CmdState.cSUB_EMPTYstart: 
				getCmdState := 'EMPTYstart';
			PTB_CmdState.cSUB_EMPTYWAITPAPERbusy: 
				getCmdState := 'EMPTYWAITPAPERbusy';
			PTB_CmdState.cSUB_EMPTYWAITPAPERGONEbusy: 
				getCmdState := 'EMPTYWAITPAPERGONEbusy';
			PTB_CmdState.cSUB_PAPERDISTANCEbusy: 
				getCmdState := 'PAPERDISTANCEbusy';
			PTB_CmdState.cSUB_PAPERDISTANCEstart: 
				getCmdState := 'PAPERDISTANCEstart';
			PTB_CmdState.cSUB_STARTENTRYDRIVE: 
				getCmdState := 'STARTENTRYDRIVE';
			PTB_CmdState.cSUB_STARTENTRYDRIVEbusy: 
				getCmdState := 'STARTENTRYDRIVEbusy';
			PTB_CmdState.cSUB_STARTSTACKDELAY: 
				getCmdState := 'STARTSTACKDELAY';
			PTB_CmdState.cSUB_WAITPAPER: 
				getCmdState := 'WAITPAPER';
			PTB_CmdState.cSUB_PAPERDISTANCESTOPbusy:
				getCmdState := 'PAPERDISTANCESTOPbusy';
		END_CASE;
	END_IF
END_IF
END_METHOD

METHOD getCtrlSIf : POINTER TO T_Ctrl_SIf_PTB
getCtrlSIf := ADR(SIf);
END_METHOD

METHOD PROTECTED IoInBridge : BOOL
// digitale and analoge inputs read from hardware or forcing
IF SIf.Cfg.bolExitSensorDebounceEnable THEN
	fbExitSensorDebounce.In_bolPresent := THIS^.In_bolBeltExitSensor;
	fbExitSensorDebounce();
	SIf.In.bolBeltExitSensor.map := fbExitSensorDebounce.Out_bolPresent;
ELSE
	SIf.In.bolBeltExitSensor.map := THIS^.In_bolBeltExitSensor;
END_IF

IF SIf.Cfg.bolEntrySensorDebounceEnable THEN
	fbEntrySensorDebounce.In_bolPresent := THIS^.In_bolBeltExitSensor;
	fbEntrySensorDebounce();
	SIf.In.bolBeltExitSensor.map := fbEntrySensorDebounce.Out_bolPresent;
ELSE
	SIf.In.bolBeltEntrySensor.map := THIS^.In_bolBeltEntrySensor;
END_IF


// Insert also an edge detection
fbPaperEntryPEdge.CLK := SIf.In.bolBeltEntrySensor.map;
fbPaperEntryPEdge();
SIf.In.bolBeltEntrySensorPEdge.map := fbPaperEntryPEdge.Q;

fbPaperEntryNEdge.CLK := SIf.In.bolBeltEntrySensor.map;
fbPaperEntryNEdge();
SIf.In.bolBeltEntrySensorNEdge.map := fbPaperEntryNEdge.Q;

fbPaperExitPEdge.CLK := SIf.In.bolBeltExitSensor.map;
fbPaperExitPEdge();
SIf.In.bolBeltExitSensorPEdge.map := fbPaperExitPEdge.Q;

fbPaperExitNEdge.CLK := SIf.In.bolBeltExitSensor.map;
fbPaperExitNEdge();
SIf.In.bolBeltExitSensorNEdge.map := fbPaperExitNEdge.Q;

IF (CIf.SwCfg.bolSimulation = FALSE) THEN
	getInBol(CIf.Job.bolIoForce,ADR(SIf.In.bolBeltExitSensor));
	getInBol(CIf.Job.bolIoForce,ADR(SIf.In.bolBeltEntrySensor));
	getInBol(CIf.Job.bolIoForce,ADR(SIf.In.bolBeltEntrySensorPEdge));
	getInBol(CIf.Job.bolIoForce,ADR(SIf.In.bolBeltEntrySensorNEdge));
	getInBol(CIf.Job.bolIoForce,ADR(SIf.In.bolBeltExitSensorPEdge));
	getInBol(CIf.Job.bolIoForce,ADR(SIf.In.bolBeltExitSensorNEdge));
ELSE
;	//simulation of global IO
END_IF
END_METHOD

METHOD PROTECTED IoOutBridge : BOOL
VAR
	bolSwitchValvesOff: BOOL;
END_VAR
// digitale and analoge inputs read from hardware or forcing
IF (CIf.SwCfg.bolSimulation = FALSE) THEN
//	setOutBol(CIf.Job.bolIoForce ,ADR(SIf.Out.intActualPosition));
;
//	THIS^.Out_intActualPosition := SIf.Out.intActualPosition.map;
END_IF
END_METHOD

METHOD PROTECTED PaperPositionHandling : BOOL
VAR_INPUT
END_VAR
// Paper Tracking Service
// -----------------------------------------------------------------------------------
CASE me.StateMachine.intState OF
	BASE_PLC.cSTA_RUN:
		fbPositionService.In_uinBeltSpeed := sif.Cur.rBeltParam.uinBeltSpeed_mms;
ELSE
	fbPositionService.In_uinBeltSpeed := 0;
END_CASE

IF SIf.In.bolBeltEntrySensorPEdge.intern THEN
	udiIdCounter := udiIdCounter + 1;
	fbPositionService.Push(udiIdCounter);
END_IF

IF SIf.In.bolBeltEntrySensorNEdge.intern THEN
	fbPositionService.EnterComplete();
END_IF

IF SIf.In.bolBeltExitSensorPEdge.intern THEN
	fbPositionService.Pop();
END_IF

// Cyclic call
fbPositionService();
SIf.Cur.uinPaperOnBelt := fbPositionService.PaperOnBelt;
END_METHOD

PROPERTY PUBLIC PositionList : POINTER TO T_PTR_STRUCT
GET
END_GET
SET
END_SET
END_PROPERTY

METHOD PROTECTED SetPumpComand : BOOL
VAR_INPUT
	intComand		: INT;
END_VAR
SetPumpComand := TRUE;

IF SIf.Cfg.bolVacuumPresent THEN
	p_fbPump^.CtrlCIf^.Job.intACmd := intComand;
END_IF
END_METHOD

METHOD PROTECTED sta_EJECTPAPER : Bool
VAR
	iDifference 		: INT;
END_VAR
// state implemetation
//--------------------------------------------------------------------------------------
// Entry action
	IF (me.StateMachine.intState<>me.StateMachine.intStateLastCycle) THEN
		me.StateMachine.intStateLastCycle := me.StateMachine.intState;
	END_IF


//--------------------------------------------------------------------------------------
// Cyclic action
	IF (me.StateMachine.intState = me.StateMachine.intStateLastCycle) THEN
		CASE me.intCmd OF
			BASE_PLC.cCMD_RUN:
				me.StateMachine.intStateNext := BASE_PLC.cSTA_RUNBusy;
			BASE_PLC.cCMD_STOP:
				me.StateMachine.intStateNext := BASE_PLC.cSTA_STOPBusy;
			PTB_CmdState.cCMD_EJECTPAPER:
				me.StateMachine.intStateNext := PTB_CmdState.cSTA_EJECTPAPERbusy;
			PTB_CmdState.cCMD_STACKPAPER:
				me.StateMachine.intStateNext := PTB_CmdState.cSTA_STACKPAPERbusy;
		END_CASE
	END_IF

//--------------------------------------------------------------------------------------
// Exit action
	IF (me.StateMachine.intState<>me.StateMachine.intStateNext) THEN
		;
	END_IF
END_METHOD

METHOD PROTECTED sta_EJECTPAPERbusy : BOOL
VAR_INPUT
END_VAR
// state implemetation
//--------------------------------------------------------------------------------------
// Entry action
	IF (me.StateMachine.intState<>me.StateMachine.intStateLastCycle) THEN
		me.StateMachine.intStateLastCycle := me.StateMachine.intState;
		cmd_RUN(sif.Par.rBeltParam.uinBeltSpeed);
		me.SubStateMachine.intStateNext := PTB_CmdState.cSUB_EMPTYWAITPAPERbusy;
	END_IF


//--------------------------------------------------------------------------------------
// Cyclic action
	IF (me.StateMachine.intState=me.StateMachine.intStateLastCycle) THEN
		CASE me.SubStateMachine.intState OF
			PTB_CmdState.cSUB_EMPTYWAITPAPERbusy:
				IF SIf.In.bolBeltExitSensor.intern THEN
					me.SubStateMachine.intStateNext := PTB_CmdState.cSUB_EMPTYWAITPAPERGONEbusy;
				END_IF
			PTB_CmdState.cSUB_EMPTYWAITPAPERGONEbusy:
				IF NOT SIf.In.bolBeltExitSensor.intern THEN
					SIf.Cur.uinPaperOnBelt := 0;
					cmd_STOP();
					me.SubStateMachine.intStateNext := PTB_CmdState.cSUB_EMPTYWAITDRIVESTOPED;
				END_IF
			PTB_CmdState.cSUB_EMPTYWAITDRIVESTOPED:
				IF (p_fbMotor^.CtrlCIf^.Job.intState = BASE_PLC.cSTA_STOP) THEN
					IF SIf.Par.bolAutoStackAfterEject THEN
						CIf.Job.intACmd := BASE_PLC.cCMD_DONE;
						CIf.Job.intMCmd := BASE_PLC.cCMD_DONE;
						me.StateMachine.intStateNext := PTB_CmdState.cSTA_STACKPAPERbusy;	
					ELSE	
						me.StateMachine.intStateNext := PTB_CmdState.cSTA_EJECTPAPER;	
					END_IF
				END_IF
		END_CASE
	END_IF


//--------------------------------------------------------------------------------------
// Exit action
	IF (me.StateMachine.intState<>me.StateMachine.intStateNext) THEN
		me.SubStateMachine.intState := BASE_PLC.cSTA_INITIALIZED;
	END_IF
END_METHOD

METHOD PROTECTED sta_ERROR : BOOL
// state implemetation
//--------------------------------------------------------------------------------------
// Entry action
	IF (me.StateMachine.intState<>me.StateMachine.intStateLastCycle) THEN
		me.StateMachine.intStateHistory := me.StateMachine.intStateLastCycle; // -> possibillity to go back to state before error
		me.StateMachine.intStateLastCycle := me.StateMachine.intState;
		pMotorCIf^.Job.intACmd := BASE_PLC.cCMD_OFF;		
	END_IF


//--------------------------------------------------------------------------------------
// Cyclic action
	IF (me.StateMachine.intState=me.StateMachine.intStateLastCycle) THEN
		
		;
		
		
		// State Change Condition
		IF (CIf.Job.bolAlmReset = TRUE) THEN
			me.StateMachine.intStateNext := cSTA_ERRORQuit;
		END_IF
	END_IF




//--------------------------------------------------------------------------------------
// Exit action
	IF (me.StateMachine.intState<>me.StateMachine.intStateNext) THEN
		;
	END_IF
END_METHOD

METHOD PROTECTED sta_ERRORQuit : BOOL
// state implemetation
//--------------------------------------------------------------------------------------
// Entry action
	IF (me.StateMachine.intState<>me.StateMachine.intStateLastCycle) THEN
		me.StateMachine.intStateLastCycle := me.StateMachine.intState;
		
	END_IF


//--------------------------------------------------------------------------------------
// Cyclic action
	IF (me.StateMachine.intState=me.StateMachine.intStateLastCycle) THEN
		
		;
		// evtl. wait time if reset of device is necessary and then decide to go to states or ERROR state
		IF (CIf.Job.bolAlmReset = TRUE) THEN
			CIf.Job.eMe_ActivAlmClass := E_AlmClass.NONE; // reset feedback channel for parent
			CIf.Job.bolAlmReset := FALSE;
		END_IF
		
		// State Change Condition
		IF (CIf.Job.bolAlmReset = FALSE) THEN
			IF (me.StateMachine.intStateHistory<=cSTA_PON) THEN
				me.StateMachine.intStateNext := cSTA_PONBusy;
			ELSIF(me.intCmd=cCMD_OFF) THEN
				me.StateMachine.intStateNext := cSTA_OFFBusy;
			ELSIF(me.intCmd=BASE_PLC.cCMD_RUN) THEN
				me.StateMachine.intStateNext := BASE_PLC.cSTA_RUNBusy;
			END_IF
		END_IF
	END_IF




//--------------------------------------------------------------------------------------
// Exit action
	IF (me.StateMachine.intState<>me.StateMachine.intStateNext) THEN
		;
	END_IF
END_METHOD

METHOD PROTECTED sta_OFF : BOOL
VAR_INPUT
END_VAR
// state implemetation
//--------------------------------------------------------------------------------------
// Entry action
	IF (me.StateMachine.intState<>me.StateMachine.intStateLastCycle) THEN
		me.StateMachine.intStateLastCycle := me.StateMachine.intState;
	END_IF


//--------------------------------------------------------------------------------------
// Cyclic action
	IF (me.StateMachine.intState=me.StateMachine.intStateLastCycle) THEN
		CASE me.intCmd OF
			BASE_PLC.cCMD_RUN:
				me.StateMachine.intStateNext := BASE_PLC.cSTA_RUNBusy;
			BASE_PLC.cCMD_STOP:
				me.StateMachine.intStateNext := BASE_PLC.cSTA_STOPBusy;
			PTB_CmdState.cCMD_EJECTPAPER:
				me.StateMachine.intStateNext := PTB_CmdState.cSTA_EJECTPAPERbusy;
			PTB_CmdState.cCMD_STACKPAPER:
				me.StateMachine.intStateNext := PTB_CmdState.cSTA_STACKPAPERbusy;
		END_CASE
	END_IF


//--------------------------------------------------------------------------------------
// Exit action
	IF (me.StateMachine.intState<>me.StateMachine.intStateNext) THEN
		;
	END_IF
END_METHOD

METHOD PROTECTED sta_OFFBusy : BOOL
VAR_INPUT
END_VAR
// state implemetation
//--------------------------------------------------------------------------------------
// Entry action
	IF (me.StateMachine.intState<>me.StateMachine.intStateLastCycle) THEN
		me.StateMachine.intStateLastCycle := me.StateMachine.intState;
		cmd_OFF();
	END_IF


//--------------------------------------------------------------------------------------
// Cyclic action
	IF (me.StateMachine.intState=me.StateMachine.intStateLastCycle) THEN

		// Set commandos not only in entry action because of possible errors or manual/auto changes
		cmd_OFF();

		IF p_fbMotor^.CtrlCIf^.Job.intState = BASE_PLC.cSTA_OFF 
		  AND CheckPumpState(BASE_PLC.cSTA_OFF) THEN
			me.StateMachine.intStateNext := BASE_PLC.cSTA_OFF;
		END_IF
	END_IF


//--------------------------------------------------------------------------------------
// Exit action
	IF (me.StateMachine.intState<>me.StateMachine.intStateNext) THEN
		;
	END_IF
END_METHOD

METHOD PROTECTED sta_PON : BOOL
VAR_INPUT
END_VAR
// state implemetation
//--------------------------------------------------------------------------------------
// Entry action
	IF (me.StateMachine.intState<>me.StateMachine.intStateLastCycle) THEN
		me.StateMachine.intStateLastCycle := me.StateMachine.intState;
		
	END_IF


//--------------------------------------------------------------------------------------
// Cyclic action
	IF (me.StateMachine.intState=me.StateMachine.intStateLastCycle) THEN
		;
	END_IF




//--------------------------------------------------------------------------------------
// Exit action
	IF (me.StateMachine.intState<>me.StateMachine.intStateNext) THEN
		;
	END_IF
END_METHOD

METHOD PROTECTED sta_RUN : Bool
VAR
	iDifference 		: INT;
END_VAR
// state implemetation
//--------------------------------------------------------------------------------------
// Entry action
	IF (me.StateMachine.intState<>me.StateMachine.intStateLastCycle) THEN
		me.StateMachine.intStateLastCycle := me.StateMachine.intState;
	END_IF


//--------------------------------------------------------------------------------------
// Cyclic action
	IF (me.StateMachine.intState = me.StateMachine.intStateLastCycle) THEN
		// The direction changed
		IF (SIf.Par.intDirection <> SIf.Cur.eActualDirection) THEN
			me.StateMachine.intStateNext := BASE_PLC.cSTA_RUNBusy;
		END_IF
		
		// The speed changed
		IF (SIf.Par.rBeltParam.uinBeltSpeed <> SIf.Cur.rBeltParam.uinBeltSpeed_mms) THEN
			me.StateMachine.intStateNext := BASE_PLC.cSTA_RUNBusy;
		END_IF
		
		IF  me.intCmd = BASE_PLC.cCMD_STOP THEN
			me.StateMachine.intStateNext := BASE_PLC.cSTA_STOPBusy;
		END_IF

		CASE SIf.Cfg.eMode OF
			E_PTB_MODE.ToDistance, 
			E_PTB_MODE.ToTime :
				IF me.StateMachine.udiTimeInState_ms > SIf.Cur.udiTimeToMove_ms THEN
					me.StateMachine.intStateNext := BASE_PLC.cSTA_STOPBusy;
				END_IF
			E_PTB_MODE.ToSensor:
				IF (SIf.In.bolBeltExitSensorPEdge.intern) THEN
					me.StateMachine.intStateNext := BASE_PLC.cSTA_STOPBusy;
				END_IF
		END_CASE
	END_IF


//--------------------------------------------------------------------------------------
// Exit action
	IF (me.StateMachine.intState<>me.StateMachine.intStateNext) THEN
		;
	END_IF
END_METHOD

METHOD PROTECTED sta_RUNBusy : BOOL
VAR_INPUT
END_VAR
// state implemetation
//--------------------------------------------------------------------------------------
// Entry action
	IF (me.StateMachine.intState<>me.StateMachine.intStateLastCycle) THEN
		me.StateMachine.intStateLastCycle := me.StateMachine.intState;
		
		CASE SIf.Cfg.eMode OF
			E_PTB_MODE.Endless,
			E_PTB_MODE.ToDistance,
			E_PTB_MODE.ToTime:
				cmd_RUN(sif.Par.rBeltParam.uinBeltSpeed);
			E_PTB_MODE.ToSensor:
				IF SIf.In.bolBeltExitSensorPEdge.intern THEN
					me.StateMachine.intStateNext := BASE_PLC.cSTA_STOPBusy;
				ELSE
					cmd_RUN(sif.Par.rBeltParam.uinBeltSpeed);
				END_IF
		END_CASE
	END_IF


//--------------------------------------------------------------------------------------
// Cyclic action
	IF (me.StateMachine.intState=me.StateMachine.intStateLastCycle) THEN
		IF (p_fbMotor^.CtrlCIf^.Job.intState = BASE_PLC.cSTA_RUN) 
		  AND (p_fbMotor^.CtrlSIf^.Cur.eDirection = arMotorDirection[SIf.Par.intDirection]) 
		  AND CheckPumpState(BASE_PLC.cSTA_RUN) THEN
			me.StateMachine.intStateNext := BASE_PLC.cSTA_RUN;
		END_IF

		IF me.intCmd = BASE_PLC.cCMD_STOP THEN
			me.StateMachine.intStateNext := BASE_PLC.cSTA_STOPBusy;
		END_IF
	END_IF


//--------------------------------------------------------------------------------------
// Exit action
	IF (me.StateMachine.intState<>me.StateMachine.intStateNext) THEN
		;
	END_IF
END_METHOD

METHOD PROTECTED sta_STACKPAPER : Bool
VAR
END_VAR
// state implemetation
//--------------------------------------------------------------------------------------
// Entry action
	IF (me.StateMachine.intState<>me.StateMachine.intStateLastCycle) THEN
		me.StateMachine.intStateLastCycle := me.StateMachine.intState;
	END_IF


//--------------------------------------------------------------------------------------
// Cyclic action
	IF (me.StateMachine.intState = me.StateMachine.intStateLastCycle) THEN
		CASE me.intCmd OF
			BASE_PLC.cCMD_RUN:
				me.StateMachine.intStateNext := BASE_PLC.cSTA_RUNBusy;
			BASE_PLC.cCMD_STOP:
				me.StateMachine.intStateNext := BASE_PLC.cSTA_STOPBusy;
			PTB_CmdState.cCMD_EJECTPAPER:
				me.StateMachine.intStateNext := PTB_CmdState.cSTA_EJECTPAPERbusy;
			PTB_CmdState.cCMD_STACKPAPER:
				me.StateMachine.intStateNext := PTB_CmdState.cSTA_STACKPAPERbusy;
		END_CASE
	END_IF


//--------------------------------------------------------------------------------------
// Exit action
	IF (me.StateMachine.intState<>me.StateMachine.intStateNext) THEN
		;
	END_IF
END_METHOD

METHOD PROTECTED sta_STACKPAPERbusy : BOOL
VAR_INPUT
END_VAR
// state implemetation
//--------------------------------------------------------------------------------------
// Entry action
	IF (me.StateMachine.intState<>me.StateMachine.intStateLastCycle) THEN
		me.StateMachine.intStateLastCycle := me.StateMachine.intState;

		me.SubStateMachine.intStateNext := PTB_CmdState.cSUB_WAITPAPER;
	END_IF


//--------------------------------------------------------------------------------------
// Cyclic action
	IF (me.StateMachine.intState=me.StateMachine.intStateLastCycle) THEN
		CASE me.SubStateMachine.intState OF
			PTB_CmdState.cSUB_WAITPAPER:
				IF SIf.In.bolBeltEntrySensor.intern THEN
					me.SubStateMachine.intStateNext := PTB_CmdState.cSUB_WAITPAPERGONE;
				ELSE
					CASE me.intCmd OF
						BASE_PLC.cCMD_RUN:
							me.StateMachine.intStateNext := BASE_PLC.cSTA_RUNBusy;
						BASE_PLC.cCMD_STOP:
							me.StateMachine.intStateNext := BASE_PLC.cSTA_STOPBusy;
						PTB_CmdState.cCMD_EJECTPAPER:
							me.StateMachine.intStateNext := PTB_CmdState.cSTA_EJECTPAPERbusy;
					END_CASE
				END_IF
			PTB_CmdState.cSUB_WAITPAPERGONE:
				IF NOT SIf.In.bolBeltEntrySensor.intern THEN
					SIf.Cur.uinPaperOnBelt := SIf.Cur.uinPaperOnBelt + 1;
					me.SubStateMachine.intStateNext := PTB_CmdState.cSUB_STARTSTACKDELAY;
				END_IF
			PTB_CmdState.cSUB_STARTSTACKDELAY:
				IF me.SubStateMachine.udiTimeInState_ms > SIf.Par.udiStackDelayTime_ms THEN
					IF SIf.Cur.uinPaperOnBelt >= SIf.Par.uinPaperStackHight THEN
						me.StateMachine.intStateNext := PTB_CmdState.cSTA_EJECTPAPERbusy;
					ELSE
						me.SubStateMachine.intStateNext := PTB_CmdState.cSUB_PAPERDISTANCEstart;
					END_IF
				END_IF
			PTB_CmdState.cSUB_PAPERDISTANCEstart:
				cmd_RUN(sif.Par.rBeltParam.uinStackSpeed);
				me.SubStateMachine.intStateNext := PTB_CmdState.cSUB_PAPERDISTANCEbusy;
			PTB_CmdState.cSUB_PAPERDISTANCEbusy:
				IF me.SubStateMachine.udiTimeInState_ms > SIf.Cur.udiTimeToMove_ms THEN
					cmd_STOP();
					me.SubStateMachine.intStateNext := PTB_CmdState.cSUB_PAPERDISTANCESTOPbusy;
				END_IF
			PTB_CmdState.cSUB_PAPERDISTANCESTOPbusy:
				IF p_fbMotor^.CtrlCIf^.Job.intState = BASE_PLC.cSTA_STOP THEN
					IF SIf.Par.bolAutoEjectAfterStack THEN
						me.StateMachine.intStateNext := PTB_CmdState.cSTA_EJECTPAPERbusy;
					ELSE
						me.StateMachine.intStateNext := PTB_CmdState.cSTA_STACKPAPER;
					END_IF
				END_IF
		END_CASE
	END_IF


//--------------------------------------------------------------------------------------
// Exit action
	IF (me.StateMachine.intState<>me.StateMachine.intStateNext) THEN
		CIf.Job.intACmd := BASE_PLC.cCMD_DONE;
		CIf.Job.intMCmd := BASE_PLC.cCMD_DONE;
		me.SubStateMachine.intState := BASE_PLC.cSTA_INITIALIZED;
	END_IF
END_METHOD

METHOD PROTECTED sta_STOP : BOOL
VAR_INPUT
END_VAR
// state implemetation
//--------------------------------------------------------------------------------------
// Entry action
	IF (me.StateMachine.intState<>me.StateMachine.intStateLastCycle) THEN
		me.StateMachine.intStateLastCycle := me.StateMachine.intState;
	END_IF


//--------------------------------------------------------------------------------------
// Cyclic action
	IF (me.StateMachine.intState=me.StateMachine.intStateLastCycle) THEN
		CASE me.intCmd OF
			BASE_PLC.cCMD_RUN:
				me.StateMachine.intStateNext := BASE_PLC.cSTA_RUNBusy;
			BASE_PLC.cCMD_STOP:
				me.StateMachine.intStateNext := BASE_PLC.cSTA_STOPBusy;
			PTB_CmdState.cCMD_EJECTPAPER:
				me.StateMachine.intStateNext := PTB_CmdState.cSTA_EJECTPAPERbusy;
			PTB_CmdState.cCMD_STACKPAPER:
				me.StateMachine.intStateNext := PTB_CmdState.cSTA_STACKPAPERbusy;
		END_CASE

		IF    (SIf.Cfg.eMode = E_PTB_MODE.ToSensor) 
		  AND (SIf.In.bolBeltExitSensorNEdge.intern) THEN
			me.StateMachine.intStateNext := BASE_PLC.cSTA_RUNBusy;
		END_IF
	END_IF


//--------------------------------------------------------------------------------------
// Exit action
	IF (me.StateMachine.intState<>me.StateMachine.intStateNext) THEN
		;
	END_IF
END_METHOD

METHOD PROTECTED sta_STOPBusy : BOOL
VAR_INPUT
END_VAR
// state implemetation
//--------------------------------------------------------------------------------------
// Entry action
	IF (me.StateMachine.intState<>me.StateMachine.intStateLastCycle) THEN
		me.StateMachine.intStateLastCycle := me.StateMachine.intState;
		cmd_STOP();
	END_IF


//--------------------------------------------------------------------------------------
// Cyclic action
	IF (me.StateMachine.intState=me.StateMachine.intStateLastCycle) THEN
		IF p_fbMotor^.CtrlCIf^.Job.intState = BASE_PLC.cSTA_STOP  THEN
			me.StateMachine.intStateNext := BASE_PLC.cSTA_STOP;
		END_IF
	END_IF


//--------------------------------------------------------------------------------------
// Exit action
	IF (me.StateMachine.intState<>me.StateMachine.intStateNext) THEN
		;
	END_IF
END_METHOD

METHOD PROTECTED StateMachine : BOOL
SUPER^.StateMachine();

// main statemachine of base controller
CASE me.StateMachine.intState OF
    BASE_PLC.cSTA_RUN: 
        THIS^.sta_RUN();
    BASE_PLC.cSTA_RUNBusy: 
        THIS^.sta_RUNBusy();
    BASE_PLC.cSTA_STOP: 
        THIS^.sta_STOP();
    BASE_PLC.cSTA_STOPBusy: 
        THIS^.sta_STOPBusy();
	PTB_CmdState.cSTA_EJECTPAPERbusy:
		THIS^.sta_EJECTPAPERbusy();
	PTB_CmdState.cSTA_EJECTPAPER:
		THIS^.sta_EJECTPAPER();
	PTB_CmdState.cSTA_STACKPAPER:
		THIS^.sta_STACKPAPER();
	PTB_CmdState.cSTA_STACKPAPERbusy:
		THIS^.sta_STACKPAPERbusy();
END_CASE;
END_METHOD

PROPERTY PUBLIC VacuumPump :  POINTER TO FB_VPC
GET
VacuumPump := p_fbPump;
END_GET
SET
p_fbPump := VacuumPump;
END_SET
END_PROPERTY

END_FUNCTION_BLOCK

// POUs/Controller/Lvl2/PBC [Paper Buffer Controller]/FB_PBC
FUNCTION_BLOCK FB_PBC EXTENDS FB_CtrlBase
VAR_INPUT
	In_bolPaperAvailableExit			: BOOL;
	In_bolPaperAvailableEntry			: BOOL;
	In_bolCapacityReached				: BOOL;
END_VAR
VAR_OUTPUT
	Out_bolAirOn						: BOOL;
END_VAR
VAR
	/// Specific interface struct for public access
	SIf									: T_Ctrl_SIf_PBC;
	///pointer to function block
	p_fbDeStacker					: POINTER TO FB_PTB;
	pDeStackerCIf					: POINTER TO BASE_PLC.T_Ctrl_CIf;
	p_fbBelt						: POINTER TO FB_PTB;
	pBeltCIf						: POINTER TO BASE_PLC.T_Ctrl_CIf;


	m_uinPaperHight_mm			: UINT := 460;
	m_uinPaperWidth_mm			: UINT := 320;
END_VAR
VAR CONSTANT
	cPAPERPOSITION_TOLERANCE_mm		: UINT := 200;
END_VAR

(*__________________________________________________________________________________________________
¦	
¦	Vistaprint Schweiz GmbH
¦	CH - 8401 Winterthur
¦
¦	www.vistaprint.ch - info@vistaprint.ch
¦___________________________________________________________________________________________________

Function desription:
Destacker/Buffer implementation. 


History:
Version		Date			Author		Comment
---------------------------------------------------------------------------------------------------
0.00.1		09.07.2013		PC			Start history
___________________________________________________________________________________________________*)


IF (me.bolActivate) THEN // cyclic call enabled
	IF (CIf.Info.bolInitDone=FALSE) THEN // first cycle -> init
		CtrlInit();
		CIf.Info.bolInitDone := TRUE;
	ELSE
		CycleStartDuty();
	
		Always();
		
		StateMachine();
		
		CycleEndDuty();
	END_IF
END_IF;

METHOD PROTECTED Always : BOOL
SUPER^.Always();

// ----------------------------------------------------------------------------------
// cyclic actions outside of statemachine
IF (me.StateMachine.intState<>cSTA_SINGLE_ANSWER) THEN
	
	; // always error supervision
	
END_IF

// ----------------------------------------------------------------------------------
// Conditions Always
IF (((me.Alarm.eActivAlmClass=E_AlmClass.EOFF) OR (me.Alarm.eActivAlmClass=E_AlmClass.OFF) OR (me.intCmd=cCMD_OFF))
		 AND (me.StateMachine.intState<>cSTA_ERROR) AND (me.StateMachine.intState<>cSTA_ERRORQuit) AND
		(me.StateMachine.intState<>cSTA_OFF) AND (me.StateMachine.intState<>cSTA_OFFBusy)) THEN
	// alarm evt EOFF, OFF or cmd off
	me.StateMachine.intStateNext := cSTA_OFFBusy;
END_IF
END_METHOD

PROPERTY PUBLIC Belt :  POINTER TO FB_PTB
GET
Belt := p_fbBelt;
END_GET
SET
p_fbBelt := Belt;
END_SET
END_PROPERTY

METHOD PROTECTED CountPaper : UINT
VAR_INPUT
END_VAR
END_METHOD

METHOD PROTECTED CtrlInit : BOOL
VAR_INPUT
END_VAR
SUPER^.CtrlInit();

pDeStackerCIf 	:= p_fbDeStacker^.CtrlCIf;
pBeltCIf 		:= p_fbBelt^.CtrlCIf;

AddChild(p_fbDeStacker^);
AddChild(p_fbBelt^);
END_METHOD

PROPERTY PUBLIC CtrlSIf : POINTER TO T_Ctrl_SIf_PBC
GET
CtrlSIf := ADR(SIf);
END_GET
SET
END_SET
END_PROPERTY

PROPERTY PUBLIC DeStacker :  POINTER TO FB_PTB
GET
DeStacker := p_fbDeStacker;
END_GET
SET
p_fbDeStacker := DeStacker;
END_SET
END_PROPERTY

